// TwinCAT 3 PLC project PLC_MOTION
// Title: PLC_MOTION_LAYER
// Author: D. Hauer
// ProjectVersion: 01.00.34
// Description: MC-PtP, NCI, Camming cyclic execution layer for motion commands
// ProgramVersion: 3.1.4026.22
// libraries:
//   Tc2_EtherCAT, * (Beckhoff Automation GmbH)
//   Tc2_MC2, * (Beckhoff Automation GmbH)
//   Tc2_MC2_Camming, * (Beckhoff Automation GmbH)
//   Tc2_MC2_Drive, * (Beckhoff Automation GmbH)
//   Tc2_MC2_FlyingSaw, * (Beckhoff Automation GmbH)
//   Tc2_MC2_XFC, * (Beckhoff Automation GmbH)
//   Tc2_NCI, * (Beckhoff Automation GmbH)
//   Tc2_PlcInterpolation, * (Beckhoff Automation GmbH)
//   Tc2_Standard, * (Beckhoff Automation GmbH)
//   Tc2_System, * (Beckhoff Automation GmbH)
//   Tc2_Utilities, * (Beckhoff Automation GmbH)
//   Tc3_Module, * (Beckhoff Automation GmbH)
// project tree:
//   CAM/ CAM.TcPOU (not stored), GVL_CAM.TcGVL (not stored)
//   CAM/class/ FB_CamAxis.TcPOU (not stored), FB_CamCtrl.TcPOU, I_Cam_Ctrl.TcIO (not stored)
//   CAM/types/ ST_CAM_CTRL.TcDUT (not stored), ST_CAM_DATA.TcDUT (not stored), ST_CAM_INFO.TcDUT (not stored), ST_CAM_READ_VALUES_PARAMETER.TcDUT (not stored), ST_CAM_STATE.TcDUT (not stored), ST_CAM_OPTIONS.TcDUT (not stored), ST_CAM_SCALING_DATA.TcDUT (not stored), ST_MOTION_FUNCTION.TcDUT (not stored), ST_MOTION_FUNCTION_POINT.TcDUT
//   FLYING_SAW/class/ FB_FlyingBase.TcPOU (not stored), FB_FlyingCtrl.TcPOU (not stored), I_Fly_Ctrl.TcIO (not stored)
//   FLYING_SAW/ FLYING_SAW.TcPOU, GVL_FLYING_SAW.TcGVL
//   FLYING_SAW/types/ ST_FLY_CTRL.TcDUT (not stored), ST_FLY_DATA.TcDUT, ST_FLY_OPTIONS.TcDUT (not stored), ST_FLY_STATE.TcDUT (not stored), ST_FLY_SYNC_MODE.TcDUT (not stored)
//   FUNCTIONS/ FUNCTIONS.TcPOU (not stored), GVL_FUNCTIONS.TcGVL (not stored)
//   FUNCTIONS/TOUCH_PROBE/ FB_TouchProbe.TcPOU (not stored), I_TouchProbe.TcIO
//   FUNCTIONS/TOUCH_PROBE/types/ ST_2BIT.TcDUT (not stored), ST_CTRL_TOUCH_PROBE.TcDUT (not stored), ST_DC_Input.TcDUT (not stored), ST_MTI_INPUT.TcDUT (not stored), ST_MTI_STATUS.TcDUT (not stored), ST_STATE_TOUCH_PROBE.TcDUT (not stored)
//   FUNCTIONS/TRIGGER_BOX/ FB_TriggerBox.TcPOU (not stored), I_TriggerBox.TcIO (not stored)
//   FUNCTIONS/TRIGGER_BOX/types/ ST_CTRL_TRIGGER.TcDUT (not stored), ST_DC_Output.TcDUT (not stored), ST_DC_State.TcDUT (not stored), ST_STATE_TRIGGER.TcDUT (not stored), T_TriggerControlBits.TcDUT (not stored)
//   MAPPING/ MAPPING_AXIS_in.TcPOU (not stored), MAPPING_AXIS_out.TcPOU (not stored)
//   MAPPING/types/ U_AXIS_CTRL.TcDUT, U_AXIS_NC_PARAMETER_WRT.TcDUT (not stored), U_AXIS_HOMING.TcDUT (not stored), U_AXIS_MOTION_OPTIONS.TcDUT (not stored), U_AXIS_MOVE_DATA.TcDUT (not stored), U_AXIS_GEAR_IN.TcDUT (not stored), U_AXIS_NC_PARAMETER_RD.TcDUT (not stored), U_AXIS_STATE.TcDUT (not stored), U_AXIS_INFO.TcDUT (not stored), U_CAM_CTRL.TcDUT (not stored), U_CAM_DATA.TcDUT, U_CAM_INFO.TcDUT (not stored), U_CAM_STATE.TcDUT (not stored), U_FLY_CTRL.TcDUT (not stored), U_FLY_DATA.TcDUT (not stored), U_FLY_OPTIONS.TcDUT (not stored), U_FLY_STATE.TcDUT (not stored), U_NCI_AXIS_ID_GROUP.TcDUT (not stored), U_NCI_CTRL.TcDUT (not stored), U_NCI_INDEX_GROUP.TcDUT, U_NCI_R_PARAMETER_I.TcDUT (not stored), U_NCI_R_PARAMETER_Q.TcDUT (not stored), U_NCI_STATE.TcDUT, U_PARAMETER_SELECTOR_CTRL.TcDUT, U_PARAMETER_SELECTOR_STATE.TcDUT (not stored), U_TOUCH_PROBE_CTRL.TcDUT (not stored), U_TOUCH_PROBE_STATE.TcDUT (not stored), U_TRIGGER_CTRL.TcDUT (not stored), U_TRIGGER_STATE.TcDUT (not stored)
//   NCI/class/ FB_NciChannel.TcPOU (not stored), FB_NciChannelCtrl.TcPOU, I_NciChannel.TcIO (not stored), I_Nci_Ctrl.TcIO (not stored)
//   NCI/ GVL_NCI.TcGVL (not stored), NCI.TcPOU
//   NCI/types/ E_NCI_CTRL.TcDUT (not stored), E_NCI_CHANNEL_ERROR.TcDUT (not stored), E_NCI_STATE.TcDUT (not stored), E_NCI_INTERPRETER_STATE.TcDUT (not stored), ST_3D_Group.TcDUT (not stored), ST_NCI_CTRL.TcDUT (not stored), ST_NCI_M_FUNC.TcDUT (not stored), ST_Index_Group.TcDUT, ST_Interface_Group.TcDUT (not stored), ST_NciChannel_Ref.TcDUT (not stored), ST_NCI_STATE.TcDUT (not stored), ST_R_Parameter.TcDUT (not stored)
//   NC_PTP/class/ FB_McAxisBase.TcPOU, FB_McAxisCtrl.TcPOU, FB_ParameterSelector.TcPOU (not stored), I_McAxis.TcIO (not stored)
//   NC_PTP/ GVL_AXIS.TcGVL (not stored), MAIN_AXIS.TcPOU
//   NC_PTP/types/axis/ E_AxisEncoderType.TcDUT (not stored), ST_HomeParams.TcDUT (not stored)
//   NC_PTP/types/control/ E_AXIS_CTRL.TcDUT (not stored), E_AXIS_SELECTOR.TcDUT (not stored), E_AXIS_STATE.TcDUT, ST_AXIS_CTRL.TcDUT (not stored), ST_AXIS_INFO.TcDUT (not stored), ST_AXIS_LIMIT_SWITCHES.TcDUT (not stored), ST_AXIS_STATE.TcDUT (not stored), ST_GEAR_IN.TcDUT (not stored), ST_HOMING.TcDUT, ST_MOTION_OPTIONS.TcDUT (not stored), ST_MOVE_DATA.TcDUT (not stored), ST_NC_PARAMETER.TcDUT (not stored), ST_PARAMETER_SELECTOR_CTRL.TcDUT (not stored), ST_PARAMETER_SELECTOR_STATE.TcDUT (not stored)
//   XFC/ FB_Xfc.TcPOU
//   XFC/types/ E_XFC_CHECK.TcDUT (not stored)
//   XTS_TRANSPORT/MSG/ GVL_MSG.TcGVL (not stored)
//   _GVL/ GlobalTextList.TcGTLO (not stored), PLC_CONSTANT.TcGVL, PLC_VERSION.TcGVL
//   _MSG/ fb_LocalTime.TcPOU, fb_MessageData.TcPOU, fb_MessageDataCtrl.TcPOU, f_MessageSet.TcPOU (not stored), GVL_MSG_AXIS.TcGVL (not stored), I_MessageData.TcIO
//   _MSG/types/ e_Device.TcDUT, E_MessageType.TcDUT (not stored), E_MESSAGE_BATCH.TcDUT, E_MESSAGE_CHECK.TcDUT (not stored), E_MESSAGE_CTRL.TcDUT (not stored), E_MESSAGE_FLOW.TcDUT (not stored), E_MESSAGE_STATE.TcDUT, e_Subdevice.TcDUT, ST_Message.TcDUT (not stored), ST_MESSAGE_CTRL.TcDUT (not stored), ST_MESSAGE_STATE.TcDUT (not stored), TL_E_MESSAGETYPE.TcTLO (not stored)
//   / PlcTask.TcTTO, Visualization Manager.TcVMO (not stored)
//   _types/ E_CHECK_STATE.TcDUT (not stored), E_PROGRESS.TcDUT (not stored), f_GetProgress.TcPOU, f_GetState.TcPOU (not stored)
// real-time tasks:
//   TASK PlcTask: cycle T#1ms, priority 20, ADS port 350
//   TASK PlcTask1: cycle T#1ms, priority 1, ADS port 351
// motion (NC):
//   TASK NC-Task 1 SAF: cycle T#2ms, priority 4, ADS port 501
//   TASK NC-Task 1 SVB: cycle T#10ms, priority 8, ADS port 511
//   AXIS Axis 1 (id 1)
//     OtherSettings: AllowMotionCmdToSlave=true
//     encoder EncType=1
//     drive DrvType=5
//       Analog: TorqueSetpointScale=10, ScaleFactorActTorque=0.1
//       TimeComp: TaskDelayCycles=1
//     controller CtrType=1
//       CtrPara: PriorControlFactor=1
//         Observer: BandWidth=20
//   AXIS Axis 2 (id 2)
//     OtherSettings: AllowMotionCmdToSlave=true
//     encoder EncType=1
//     drive DrvType=5
//       Analog: TorqueSetpointScale=10, ScaleFactorActTorque=0.1
//       TimeComp: TaskDelayCycles=1
//     controller CtrType=1
//       CtrPara: PriorControlFactor=1
//         Observer: BandWidth=20
//   AXIS Axis 3 (id 3)
//     OtherSettings: AllowMotionCmdToSlave=true
//     encoder EncType=1
//     drive DrvType=5
//       Analog: TorqueSetpointScale=10, ScaleFactorActTorque=0.1
//       TimeComp: TaskDelayCycles=1
//     controller CtrType=1
//       CtrPara: PriorControlFactor=1
//         Observer: BandWidth=20
//   AXIS Axis 4 (id 4)
//     OtherSettings: AllowMotionCmdToSlave=true
//     encoder EncType=1
//     drive DrvType=5
//       Analog: TorqueSetpointScale=10, ScaleFactorActTorque=0.1
//       TimeComp: TaskDelayCycles=1
//     controller CtrType=1
//       CtrPara: PriorControlFactor=1
//         Observer: BandWidth=20
//   AXIS Axis 5 (id 5)
//     OtherSettings: AllowMotionCmdToSlave=true
//     encoder EncType=1
//     drive DrvType=5
//       Analog: TorqueSetpointScale=10, ScaleFactorActTorque=0.1
//       TimeComp: TaskDelayCycles=1
//     controller CtrType=1
//       CtrPara: PriorControlFactor=1
//         Observer: BandWidth=20
//   AXIS Axis 6 (id 6)
//     OtherSettings: AllowMotionCmdToSlave=true
//     encoder EncType=1
//     drive DrvType=5
//       Analog: TorqueSetpointScale=10, ScaleFactorActTorque=0.1
//       TimeComp: TaskDelayCycles=1
//     controller CtrType=1
//       CtrPara: PriorControlFactor=1
//         Observer: BandWidth=20
// variable links:
//   ExternControl/ExternControl Instance <-> PLC_MOTION/PLC_MOTION Instance
//     PlcTask Inputs/MAIN.eInitPlcMotion <-> PlcTask Outputs/MAIN_AXIS.eInit
//     PlcTask Inputs/MAPPING_in.AxisInfo.byState <-> PlcTask Outputs/MAPPING_AXIS_out.AxisInfo.byState
//     PlcTask Inputs/MAPPING_in.AxisParameterRd.byState <-> PlcTask Outputs/MAPPING_AXIS_out.AxisParameterOut.byState
//     PlcTask Inputs/MAPPING_in.AxisState.byState <-> PlcTask Outputs/MAPPING_AXIS_out.AxisState.byState
//     PlcTask Outputs/MAPPING_out.AxisCtrl.byCtrl <-> PlcTask Inputs/MAPPING_AXIS_in.AxisCtrl.byCtrl
//     PlcTask Outputs/MAPPING_out.AxisGearInData.byCtrl <-> PlcTask Inputs/MAPPING_AXIS_in.AxisGearInData.byCtrl
//     PlcTask Outputs/MAPPING_out.AxisHoming.byCtrl <-> PlcTask Inputs/MAPPING_AXIS_in.AxisHoming.byCtrl
//     PlcTask Outputs/MAPPING_out.AxisMotionOptions.byCtrl <-> PlcTask Inputs/MAPPING_AXIS_in.AxisMotionOptions.byCtrl
//     PlcTask Outputs/MAPPING_out.AxisMoveData.byCtrl <-> PlcTask Inputs/MAPPING_AXIS_in.AxisMoveData.byCtrl
//     PlcTask Outputs/MAPPING_out.AxisParameterWrt.byCtrl <-> PlcTask Inputs/MAPPING_AXIS_in.AxisParameterIn.byCtrl
//   PLC_MOTION/PLC_MOTION Instance <-> NC-Task 1 SAF/Axes/Axis 1
//     PlcTask Inputs/GVL_AXIS.AxisRef[1].NcToPlc <-> Outputs/ToPlc
//     PlcTask Outputs/GVL_AXIS.AxisRef[1].PlcToNc <-> Inputs/FromPlc
//   PLC_MOTION/PLC_MOTION Instance <-> NC-Task 1 SAF/Axes/Axis 2
//     PlcTask Inputs/GVL_AXIS.AxisRef[2].NcToPlc <-> Outputs/ToPlc
//     PlcTask Outputs/GVL_AXIS.AxisRef[2].PlcToNc <-> Inputs/FromPlc
//   PLC_MOTION/PLC_MOTION Instance <-> NC-Task 1 SAF/Axes/Axis 3
//     PlcTask Inputs/GVL_AXIS.AxisRef[3].NcToPlc <-> Outputs/ToPlc
//     PlcTask Outputs/GVL_AXIS.AxisRef[3].PlcToNc <-> Inputs/FromPlc
//   PLC_MOTION/PLC_MOTION Instance <-> NC-Task 1 SAF/Axes/Axis 4
//     PlcTask Inputs/GVL_AXIS.AxisRef[4].NcToPlc <-> Outputs/ToPlc
//     PlcTask Outputs/GVL_AXIS.AxisRef[4].PlcToNc <-> Inputs/FromPlc
//   PLC_MOTION/PLC_MOTION Instance <-> NC-Task 1 SAF/Axes/Axis 5
//     PlcTask Inputs/GVL_AXIS.AxisRef[5].NcToPlc <-> Outputs/ToPlc
//     PlcTask Outputs/GVL_AXIS.AxisRef[5].PlcToNc <-> Inputs/FromPlc
//   PLC_MOTION/PLC_MOTION Instance <-> NC-Task 1 SAF/Axes/Axis 6
//     PlcTask Inputs/GVL_AXIS.AxisRef[6].NcToPlc <-> Outputs/ToPlc
//     PlcTask Outputs/GVL_AXIS.AxisRef[6].PlcToNc <-> Inputs/FromPlc

CONFIGURATION PLC_MOTION
    RESOURCE PLC ON TwinCAT3
        TASK PlcTask(INTERVAL := T#1ms, PRIORITY := 1);
        PROGRAM MAPPING_AXIS_in WITH PlcTask : MAPPING_AXIS_in;
        PROGRAM MAIN_AXIS WITH PlcTask : MAIN_AXIS;
        PROGRAM FUNCTIONS WITH PlcTask : FUNCTIONS;
        PROGRAM NCI WITH PlcTask : NCI;
        PROGRAM CAM WITH PlcTask : CAM;
        PROGRAM FLYING_SAW WITH PlcTask : FLYING_SAW;
        PROGRAM MAPPING_AXIS_out WITH PlcTask : MAPPING_AXIS_out;
    END_RESOURCE
END_CONFIGURATION

// ---- CAM/types/ST_MOTION_FUNCTION_POINT.TcDUT
{attribute 'pack_mode' := '2'}
TYPE ST_MOTION_FUNCTION_POINT :
STRUCT
   nPointIndex            : UINT;
   nFunctionType          : UINT;
   wPointType             : WORD;
   nRelIndexNextPoint     : UINT;
   rMasterPos             : LREAL; (* X *)
   rSlavePos              : LREAL; (* Y *)
   rSlaveVelo             : LREAL; (* Y' *)
   rSlaveAcc              : LREAL; (* Y'' *)
   rSlaveJerk             : LREAL; (* Y''' *)
END_STRUCT
END_TYPE

// ---- FLYING_SAW/types/ST_FLY_DATA.TcDUT
{attribute 'pack_mode' := '2'}
TYPE ST_FLY_DATA :
STRUCT
  rDeltaToMasterPos       : LREAL;
  rModuloSyncPosSlave     : LREAL;
  rMasterStartDistance    : LREAL;
  rDelta                  : LREAL  := 0.1;
  rGearNumerator          : LREAL;
  iGearDenumerator        : USINT  := 1;
  nMasterAxisId           : UDINT; // NC axis ID, index is looked up by Cmd
  rModulo                 : lreal; // float for modulo calculation, this is independent of the NC on purpose, you may connect the modulo divisor from the NC on the outside of the FlyingSaw class
END_STRUCT
END_TYPE

// ---- MAPPING/types/U_AXIS_CTRL.TcDUT
TYPE U_AXIS_CTRL :
UNION

  stCtrl              : ARRAY[1..MAX_AXIS] OF ST_AXIS_CTRL;

  byCtrl    AT %I*    : ARRAY[1..MAX_AXIS] OF
                        ARRAY[1..SIZEOF(ST_AXIS_CTRL)] OF BYTE;
END_UNION
END_TYPE

// ---- MAPPING/types/U_CAM_DATA.TcDUT
TYPE U_CAM_DATA :
UNION
  stCtrl              : ARRAY[1..MAX_AXIS] OF ST_CAM_DATA;

  byCtrl    AT %I*    : ARRAY[1..MAX_AXIS] OF
                        ARRAY[1..SIZEOF(ST_CAM_DATA)] OF BYTE;
END_UNION
END_TYPE

// ---- MAPPING/types/U_NCI_INDEX_GROUP.TcDUT
TYPE U_NCI_INDEX_GROUP :
UNION

  stCtrl              : ARRAY[1..MAX_NCI_CH] OF ST_Index_Group;

  byCtrl    AT %I*    : ARRAY[1..MAX_NCI_CH] OF
                        ARRAY[1..SIZEOF(ST_Index_Group)] OF BYTE;
END_UNION
END_TYPE

// ---- MAPPING/types/U_NCI_STATE.TcDUT
TYPE U_NCI_STATE :
UNION

  stState             : ARRAY[1..MAX_NCI_CH] OF ST_NCI_STATE;

  byState   AT %Q*    : ARRAY[1..MAX_NCI_CH] OF
                        ARRAY[1..SIZEOF(ST_NCI_STATE)] OF BYTE;
END_UNION
END_TYPE

// ---- MAPPING/types/U_PARAMETER_SELECTOR_CTRL.TcDUT
TYPE U_PARAMETER_SELECTOR_CTRL :
UNION
  stCtrl              : ST_PARAMETER_SELECTOR_CTRL;

  byCtrl    AT %I*    : ARRAY[1..SIZEOF(ST_PARAMETER_SELECTOR_CTRL)] OF BYTE;

END_UNION
END_TYPE

// ---- NCI/types/ST_Index_Group.TcDUT
{attribute 'pack_mode' := '2'}
TYPE ST_Index_Group :
STRUCT
  nXAxisIdx     : UDINT := 1;
  nYAxisIdx     : UDINT := 2;
  nZAxisIdx     : UDINT := 3;

  nQ1AxisIdx    : UDINT;
  nQ2AxisIdx    : UDINT;
  nQ3AxisIdx    : UDINT;
  nQ4AxisIdx    : UDINT;
  nQ5AxisIdx    : UDINT;
END_STRUCT
END_TYPE

// ---- NC_PTP/types/control/E_AXIS_STATE.TcDUT
{attribute 'qualified_only'}
{attribute 'to_string'}
TYPE E_AXIS_STATE :
(
  AXIS_NULL,   // null reaction to command
  AXIS_INIT,
  AXIS_DISABLE,
  AXIS_ENABLE,

  AXIS_NO_INIT  := 9,
  
  AXIS_IDLE     := 10, // clear axis and enable
  AXIS_HOME,
  AXIS_MOVE_POS,
  AXIS_MOVE_VELO,
  AXIS_HALT,
  AXIS_STOP,
  AXIS_SEND_TO_POS,

  AXIS_RESET              := 19,
  AXIS_STARTUP            := 20,

  AXIS_MOVE_BUFFER        := 30,
  AXIS_MOVE_BUFFER_VELO,

  AXIS_PARAMETER_READ     := 40, // command for reading and writing parameter
  AXIS_PARAMETER_WRITE,
  AXIS_PARAMETER_WRITE_PERSISTENT,


  AXIS_GEAR_IN            := 50,
  AXIS_GEAR_OUT,
  AXIS_GEAR_IN_MULTIMASTER,

  CAM_INIT                := 60,
  CAM_IN,
  CAM_OUT,
  CAM_SCALING,
  CAM_INFO,
  CAM_RD_MOTION_FUNCTION,
  CAM_RD_MOTION_FUNCTION_POINT,
  CAM_RD_MOTION_FUNCTIONS_VALUES,
  CAM_WRT_MOTION_FUNCTION,
  CAM_WRT_MOTION_FUNCTION_POINT

)UINT;
END_TYPE

// ---- NC_PTP/types/control/ST_HOMING.TcDUT
{attribute 'pack_mode' := '2'}
TYPE ST_HOMING :
STRUCT
  bExecute      : BIT;

  stHomingParam : ST_HomeParams;
END_STRUCT
END_TYPE

// ---- _MSG/types/e_Device.TcDUT
{attribute 'to_string'}
TYPE e_Device :
(
  // txt file logging LOG_FILE
  Device_Null,                  // NULL               - not to be used
  Device_Main,                  // MAIN(PRG)          - reserved for MAIN(PRG)
  Device_Nci,                   // NCI(PRG)           - reserved for NCI(PRG)
  Device_Cam,                   // CAM(PRG            - reserved for CAM(PRG)
  Device_Functions,             // FUNCTIONS(PRG)     - reserved for FUNCTIONS(PRG)
  Device_FlyingSaw,             // FLYING_SAW(PRG)    - reserved for FLYING_SAW(PRG)
  Device_MainApplication,       // MAIN_APP(PRG)

  Device_ParameterSelector,     // fb_ParameterSelector can only exist once in a project.
  Device_Configuration,         // fb_Configuration can handle multiple files therefore only one instance is required
  Device_XmlData,               // generic XML Data (e.g. persistent data)
  Device_Utilities,             // service calls to anyone you may want to talk to, the main intent is to get XPU and TcXtsIo data to the application side


  General           :=  1000,
  CaGroup           :=  2000,
  Xpu               :=  3000,
  XpuCtrl           :=  4000,
  Mover             :=  5000,
  MoverCtrl         :=  6000,
  XtsTransportUnit  :=  7000,
  XfcTriggerBox     :=  8000,
  XfcTouchProbe     :=  9000,
  XtsStation        := 10000,

  Camming           := 11000,
  NciChannel        := 12000,
  NciChannelCtrl    := 13000,
  Axis              := 14000,
  XfcAxis           := 15000,

  // txt file logging LOG_FILE_METRICS
  Metrics           := 16000,

  FlyingSaw         := 17000,


  // txt file logging LOG_FILE_APP
  Process           := 20000,
  ProcessListCtrl   := 21000,
  TicketListCtrl    := 22000,

  Application       := 30000,

  // txt file logging LOG_FILE_PRODUCT - this is for you to use
  DataProduct       := 40000
)UDINT;
END_TYPE

// ---- _MSG/types/E_MESSAGE_BATCH.TcDUT
{attribute 'qualified_only'}
{attribute 'strict'}
{attribute 'to_string'}
TYPE E_MESSAGE_BATCH :
(
	MSG_BATCH_NULL,
  MSG_BATCH_JOB_STARTED,
  MSG_BATCH_NEXT_IN_JOB,
  MSG_BATCH_JOB_DONE
)UINT;
END_TYPE

// ---- _MSG/types/E_MESSAGE_STATE.TcDUT
{attribute 'qualified_only'}
//{attribute 'strict'}
{attribute 'to_string'}
TYPE E_MESSAGE_STATE :
(
	MSG_STATE_NULL,
  MSG_STATE_INIT    := 10,
  MSG_STATE_IDLE    := 30,
  MSG_STATE_WRITE   := 50
)UINT;
END_TYPE

// ---- _MSG/types/e_Subdevice.TcDUT
{attribute 'strict'}
{attribute 'to_string'}
TYPE e_Subdevice :
(
  // sub device for message system
  General                 :=  0,
  MainInit,
  // Motion Control FB Instances
  fbPower,
  fbReset,
  fbResetSercos,
  fbHalt,
  fbStop,                 // 5
  fbHome,
  fbJog,
  fbMoveVelocity1,
  fbMoveVelocity2,
  fbMoveAbsolute1,        // 10
  fbMoveAbsolute2,
  fbMoveEndless,
  fbMovePtP,
  fbMoveVelo,

  // CA CollisionAvoidance FB instances
  // CA group fb instances
  fbCaGroup             := 30,
  fbMoveToPosCa,
  fbSendToAbsPosCa,
  fbSendToModuloPosCa,
  fbGearInPosCa,
  fbGroupAddAxis,
  fbGroupRemoveAxis,
  fbGroupDisable,
  fbGroupEnable,
  fbGroupErrorRead,
  fbGroupStatusRead,
  fbGroupReset,
  fbGroupStop,
  fbHaltCa,
  fbSendToPos,

  fbGearIn                := 50,
  fbGearOut,
  fbGearInMultiMaster,

  fbGearInPos,
  fbGearInVelo,


  fbCamOut                := 80,
  fbCamInV2,
  fbCamScalingV2,
  fbCamInfoV2,
  fbReadMotionFunction,
  fbReadMotionFunctionPoint,
  fbReadMotionFunctionValues,
  fbWriteMotionFunction,
  fbWriteMotionFunctionPoint,
  fbSetOnlineChangeMode,

  fbReadParameter         := 100,
  fbReadBoolParameter,
  fbWriteParameter,
  fbWriteBoolParameter,
  fbWriteParameterPersistent,

  fbBuildGroup            := 200,
  fbClearGroup,
  fbLoadProg,
  fbResetItp,
  fbStartStopItp,
  fbEStopItp,             // 205
  fbStepOnAfterEStopItp,
  fbConfirmHskItp,
  fbDelDtgItp,
  fbNciFeedTablePreparation,
  fbNciFeedTable,         // 210
  fbReadLine,
  fbItpReadRParams,
  fbItpWriteRParams,
  Get_ItpState,
  Get_Error,              // 215


  XfcPositionAtTime       := 300,
  XfcTimeOfPosition,
  XfcTimeToPosition,
  XfcTimeToModuloPosition,
  XfcRecordedPosition,
  XfcTouchProbe,          // 305
  XfcTouchProbeEL1258,
  XfcTouchProbeOptions,
  XfcTriggerRef,
  XfcTriggerRef_MT,
  XfcEl1258Interface_MT,  // 310
  XfcRecordedPosition_MT,
  XfcTriggerOut,
  XfcTriggerStart,
  XfcSwitchOn_2252,
  XfcSwitchOff_2252,      // 315
  XfcInit,
  XfcLatchPosition,
  XfcWaitForPosition,

  AxisMode              := 1000,
  AxisControl,
  AxisStartUp,
  AxisCycle,
  AxisIdle,

  NciControl            := 2000,
  NciStartUp,
  NciCycle,
  NciIdle,

  FlyingSawControl      := 2100,
  FlyingSawStartUp,


  StationLinkedList     := 3000,
  StationInitList,
  StationAddHead,
  StationAddTail,
  StationGetHead,
  StationRemoveHeadValue,
  StationGearInDistanceToSync,
  StationGearInSyncStart,
  StationGearInSyncMove,
  StationGearInSyncEnd,
  StationCalcInfeedPosition,

  StationControl        := 4000,
  StationState, 

  Xpu_fbEnvironment     := 5000,
  Xpu_fbProcessingUnit,
  Xpu_fbXpuPart,
  Xpu_fbXpuTrack,
  Xpu_fbMc2CaGroup,
  Xpu_fbParameterSet,
  Xpu_fbNctController,

  Xpu_fbPartModules     := 5500,

  Xpu_fbMoverXpu        := 6000,

  Xpu_fbNctBaseUnit     := 6500,

  TransportUnit_General := 7000,
  TransportUnit_Restart := 7010,
  TransportUnit_Start,
  TransportUnit_XpuInit,
  TransportUnit_StationClearOutfeed,

  CamControl            := 8000,
  CamStartUp,
  CamCycle,

  Process_StationCollector    := 11000,
  Process_ProcessCollector    := 11100,
  Process_ProcessCollector_Init,
  Process_ProcessCollector_Cycle,
  Process_ProcessCollector_Control,

  Process_LinkedList_GetHead,
  Process_LinkedList_RemoveHead,
  Process_LinkedList_AddTail,
  Process_LinkedList_CheckData,
  Process_StationQueue_Check,

  Process_LinkedList_Com              := 11200,
  Process_LinkedList_Com_Init,
  Process_LinkedList_Com_Cmd,
  Process_LinkedList_Com_AddHead,
  Process_LinkedList_Com_AddTail,
  Process_LinkedList_Com_DelHead,
  Process_LinkedList_Com_DelTail,
  Process_LinkedList_Com_GetHead,
  Process_LinkedList_Com_GetTail,


  Instance_Command              := 12000,
  Instance_ProcessConductor,
  Instance_BufferInfeed,
  Instance_Infeed,
  Instance_BufferOutfeed,
  Instance_Outfeed,
  Instance_Sender_Buffer,

  Ticket_LinkedList_Ctrl        := 12100,
  Ticket_LinkedList_Com_Init,
  Ticket_LinkedList_Com_Cmd,
  Ticket_LinkedList_Com_AddHead,
  Ticket_LinkedList_Com_AddTail,
  Ticket_LinkedList_Com_DelHead,
  Ticket_LinkedList_Com_DelTail,
  Ticket_LinkedList_Com_GetHead,
  Ticket_LinkedList_Com_GetTail,
  

  Application                 := 13000,
  Application_Check,
  Application_Clear,
  Application_Cmd,
  Application_Disable,
  Application_Enable,
  Application_Finish,
  Application_Init,
  Application_Proceed,
  Application_Work


)DINT;
END_TYPE

// ---- FLYING_SAW/GVL_FLYING_SAW.TcGVL
{attribute 'qualified_only'}
VAR_GLOBAL
  //-----------------------------------------------------------------------------
  // command and state structure
  //  - datafields for anyone to access
  //    - ADS via symbol
  //    - cyclic mapping to any other cyclic network/runtime
  //-----------------------------------------------------------------------------
  Ctrl                        : ARRAY[1..PLC_CONSTANT.MAX_AXIS] OF ST_FLY_CTRL;      // command structure to write into
  State                       : ARRAY[1..PLC_CONSTANT.MAX_AXIS] OF ST_FLY_STATE;     // state structure to read from


  //-----------------------------------------------------------------------------
  // data and info structure
  //  - parameter data fields for
  //    - Ctrl  --> Data
  //    - State --> Info
  //-----------------------------------------------------------------------------
//  Info                        : ARRAY[1..PLC_CONSTANT.MAX_AXIS] OF ST_FLY_INFO;
  Data                        : ARRAY[1..PLC_CONSTANT.MAX_AXIS] OF ST_FLY_DATA;


  //-----------------------------------------------------------------------------
  // R/W datafields
  // - optional data for CheckMask
  // - The Options contains two position values as limits. 
  //   The check for these position limits can be activated. 
  //   To do this, two flags 
  //   (GearInSync_CheckMask_OptionalMinPos, 
  //    GearInSync_CheckMask_OptionalMaxPos) 
  //   have to be set in the SyncMode structure.
  //
  //-----------------------------------------------------------------------------
  Options                     : ARRAY[1..PLC_CONSTANT.MAX_AXIS] OF ST_FLY_OPTIONS;


  //-----------------------------------------------------------------------------
  // cyclic interface function block: FB_FlyingCtrl
  //  - Tc2_MC2_FlyingSaw functions are here 
  //-----------------------------------------------------------------------------
{IF defined (SAW)}
  {info 'PLC_MOTION_LAYER: FLYING_SAW'}
  Control                     : ARRAY[1..PLC_CONSTANT.MAX_AXIS] OF FB_FlyingCtrl;
{ELSE}
  Control                     : ARRAY[1..PLC_CONSTANT.MAX_AXIS] OF I_Fly_Ctrl;
{END_IF}

END_VAR

// ---- _GVL/PLC_CONSTANT.TcGVL
//{attribute 'qualified_only'}
VAR_GLOBAL CONSTANT


  //-----------------------------------------------------------------------------
  // AXIS related limits
  //-----------------------------------------------------------------------------
  MAX_AXIS              : UINT    := 6;
  MAX_RETRY             : UINT    := 5;


  //-----------------------------------------------------------------------------
  // NCI related limits and *.nc standard folder
  //-----------------------------------------------------------------------------
{IF NOT defined (BSD)}
  NCI_DIR               : STRING  := 'C:\TwinCAT\Mc\Nci\';
{ELSE}
  NCI_DIR               : STRING  := '/usr/local/etc/TwinCAT/Mc/Nci/';
{END_IF}

{IF defined (NCI)}
  {info 'PLC_MOTION_LAYER: NCI'}
  NCI_ACTIVE            : BOOL    := TRUE;
  CONFIG_NAME           : STRING  := 'NCI_Spec_Ch_';
{ELSE}
  NCI_ACTIVE            : BOOL    := FALSE;
  CONFIG_NAME           : STRING  := 'NCI_NOT_ACTIVE';
{END_IF}

  MAX_NCI_CH            : UINT    := 1;

  MAX_PATH_STEPS        : UINT    := 5;
  MAX_MC_AXIS           : UINT    := 3;
  MAX_AUX_AXIS          : UINT    := 2;
  MAX_R_PARA            : UINT    := 10;


  //-----------------------------------------------------------------------------
  // CAMMING related limits
  //-----------------------------------------------------------------------------
{IF defined (CAM)}
  {info 'PLC_MOTION_LAYER: CAM'}
  CAM_ACTIVE                  : BOOL    := TRUE;
{ELSE}
  CAM_ACTIVE                  : BOOL    := FALSE;
{END_IF}

  MAX_CAM_CH                  : UINT    := 1;

  MAX_MOTION_FUNCTION_POINTS  : UINT    := 10;

  // HAUD
  // 17.07.2024
  // Start Implementation of Position Trigger function
  //  - Timestamp/position output
  //  - Latch DC time from input
  
  MAX_TRIGGER_BOX             : UINT := 12;
  MAX_TOUCH_PROBE             : UINT := 12;
  MAX_TRIGGER_COUNT           : UINT :=  4;
  MAX_MTI_CH                  : UINT :=  1; // MAX mti channel per EL terminal

{IF defined (XFC)}
  {info 'PLC_MOTION_LAYER: XFC'}
  XFC_ACTIVE                  : BOOL := TRUE;
{ELSE}
  XFC_ACTIVE                  : BOOL := FALSE;
{END_IF}

  // HAUD
  // 2026 05 28
  // Gear In Pos implementation for flying saw application 

{IF defined (SAW)}
  {info 'PLC_MOTION_LAYER: FLYING_SAW'}
  FLY_SAW_ACTIVE              : BOOL  := TRUE;
{ELSE}
  FLY_SAW_ACTIVE              : BOOL  := FALSE;
{END_IF}
END_VAR

// ---- _GVL/PLC_VERSION.TcGVL
{attribute 'qualified_only'}
VAR_GLOBAL CONSTANT
  VERSION               : STRING := 'V 01.00.38';

  // 2025 05 28 HAUD
  // Flying Saw wrapper

  // 2025 05 13 HAUD
  //
  // FB_McAxisBase.MoveVeloBuffer Test, changes for setpoint change detection

  // 2025 10 24 HAUD
  //
  // documentation added, 
  // project dev changed to 4026.19
  // Ambiguities resoved

  // 2025 08 21 HAUD
  //
  // e_Device: Application added
  // e_Subdevices: merge with XTS_TRANSPORT_LAYER
  // FB_McAxis: testing SendToPos, distance added to method interface

  // 2025 02 17 HAUD
  //
  // code review
  // Message Levels are set during initialization
  // sizeof mapping data is fetched at startup only

  // 2025 01 09 HAUD
  //
  // - FUNCTIONS
  //    - code review
  //    - ctrl/state mechanic harmonized
  // - MAPPING
  //    - UNIONS added

  // 2024 08 08 HAUD
  //
  // - TC_PLC_MOTION_LAYER: 
  //    - XFC base class added
  //    - TriggerBox (DC output set, DC Input latch)
  //    - TouchProbe (DC Input latch: positive, negative)

  // 2024 06 21 HAUD
  //
  // - TC_PLC_MOTION_LAYER: 
  //    - E_PROGRESS refactoring to match TC_XTS_TRANSPORT_LAYER
  

  // 2024 06 10 HAUD
  //
  // - TC_PLC_MOTION_LAYER: 
  //    - rename repository
  //    - remove LEGACY compatibility
  //
  // - PLC_OPEN_DRIVE:
  //    - deprecated


  // 2024 05 31 HAUD
  // 
  // V 01.00.02
  // precompiler defines: 
  //  - BSD: 
  //    - Tc-BSD file system is used else Windows file system is used
  //
  //  - TEST:
  //    - GVL_MSG.MessageLevel
  // Axis, Cam, Nci have individual message levels now

  // 2024 03 09 HAUD
  // 
  // V 01.00.01
  // MC PtP - execution layer with optional mapping
  // NCI    - execution layer with optional mapping
  // CAM    . execution layer with optional mapping
  // precompiler defines: 
  //  - WIN: windows file system is used else Tc-BSD file system is used
  //  - NCI: NCI libraries are linked in project
  //  - CAM: Camming libraries are linked in project
  //  - AXIS_MAP: mapping is used


  // 2024 02 15 HAUD
  // 
  // V 00.50.04
  //
  // Buffered moves test
  // CamIn Test --> TODO MultiCam
  // Message system, cyclic check for write
  

  // 2024 01 12 HAUD
  //
  // V 00.50.03
  //
  // Building is done
  // start of UnitTesting

  // 2024 01 17 HAUD
  //
  // V 00.50.02
  // 
  // start camming implementation (MC_CamIn_V2)
  // legacy namespace available for downward compatibility of ADS Symbol names

  // 2023 12 23 HAUD
  // NC_PTP
  // - redesign for PLC_OPEN_DRIVE started 
  //    --> E_PROGRESS for state feedback
  // - FB_AxisControl inherits FB_McAxis


  //  2023 10 19
  //  HAUD
  // first draft 
  // TODO: everything

END_VAR

// ---- FUNCTIONS/TOUCH_PROBE/I_TouchProbe.TcIO
INTERFACE I_TouchProbe

PROPERTY Ctrl : REFERENCE TO ARRAY [1..MAX_TOUCH_PROBE] OF ST_CTRL_TOUCH_PROBE
SET
END_SET
END_PROPERTY

METHOD Cycle : BOOL
VAR_INPUT
END_VAR
END_METHOD

PROPERTY Index : udint
GET
END_GET
SET
END_SET
END_PROPERTY

PROPERTY Input : pointer TO ARRAY [1..MAX_TOUCH_PROBE] OF ST_MTI_Input
SET
END_SET
END_PROPERTY

PROPERTY InputState : pointer TO ARRAY [1..MAX_TOUCH_PROBE] OF ST_MTI_STATUS
SET
END_SET
END_PROPERTY

PROPERTY ItfAxis : ARRAY[1..MAX_AXIS]       OF I_McAxis
SET
END_SET
END_PROPERTY

PROPERTY MessageLevel : e_messagetype
GET
END_GET
SET
END_SET
END_PROPERTY

PROPERTY State :  REFERENCE TO ARRAY[1..MAX_TOUCH_PROBE] OF ST_STATE_TOUCH_PROBE;
SET
END_SET
END_PROPERTY

END_INTERFACE

// ---- _MSG/I_MessageData.TcIO
INTERFACE I_MessageData

PROPERTY DirRoot : POINTER to string(255)
SET
END_SET
END_PROPERTY

PROPERTY ErrorIndex : reference to uint
SET
END_SET
END_PROPERTY

PROPERTY FileRoot : pointer to string(255)
SET
END_SET
END_PROPERTY

PROPERTY LocalTime : pointer to DT
SET
END_SET
END_PROPERTY

PROPERTY MessageIndex : reference to uint
SET
END_SET
END_PROPERTY

PROPERTY MsgList : pointer to ARRAY[1..GVL_MSG.MAX_MESSAGE] OF st_message
SET
END_SET
END_PROPERTY

END_INTERFACE

// ---- NC_PTP/MAIN_AXIS.TcPOU
PROGRAM MAIN_AXIS
VAR
  eInit         AT %Q*      : E_PROGRESS;   // shall be checked by controlling entity, before using Ctrl/State structs

  nAxis,
  nAxisInit                 : UINT;

  stMsg                   : ST_Message;
  eMsgState               : e_message_state;
  eMsgProgress            : E_PROGRESS;
  eMtrState               : e_message_state;
  eMtrProgress            : E_PROGRESS;

  tIdleWriteMotion        : TIME := T#5S;
  tIdleWriteMetric        : TIME := T#5S;
  tonIdleWriteMotion      : Tc2_Standard.TON;
  tonIdleWriteMetric      : Tc2_Standard.TON;
END_VAR

//-----------------------------------------------------------------------------------------------------------------
// Local time; used for timestamps
//-----------------------------------------------------------------------------------------------------------------
GVL_MSG_AXIS.fbLocalTime();
GVL_MSG.sLocalTime                            :=
GVL_MSG_AXIS.sLocalTime                       := GVL_MSG_AXIS.fbLocalTime.LocalTimeString;
GVL_MSG.dtLocalTime                           :=
GVL_MSG_AXIS.dtLocalTime                      := GVL_MSG_AXIS.fbLocalTime.LocalTime;
//-----------------------------------------------------------------------------------------------------------------
// /assign dataflow
//-----------------------------------------------------------------------------------------------------------------
FOR nAxis := 1 TO PLC_CONSTANT.MAX_AXIS
DO
  GVL_AXIS.Control[nAxis].AxisIndex           := nAxis;
  GVL_AXIS.Control[nAxis].MessageLevel        := GVL_MSG_AXIS.MessageLevelAxisPtp[nAxis];

  GVL_AXIS.Control[nAxis].AxisCtrl            := ADR(GVL_AXIS.Ctrl);          // command
  GVL_AXIS.Control[nAxis].AxisState           := ADR(GVL_AXIS.State);         // state + result of command

  GVL_AXIS.Control[nAxis].Axes                REF=   GVL_AXIS.AxisRef;        // All for one; coupling requires access across all axes

  GVL_AXIS.Control[nAxis].AxisInfo            := ADR(GVL_AXIS.Info);          // axis information: act/set values and bits from axis
  GVL_AXIS.Control[nAxis].AxisData            := ADR(GVL_AXIS.Data);          // position and dynamic constraints for movement
  GVL_AXIS.Control[nAxis].AxisGearInParameter := ADR(GVL_AXIS.GearInParameter);

  GVL_AXIS.Control[nAxis].NcParameterOut      := ADR(GVL_AXIS.NcParameterOut);
  GVL_AXIS.Control[nAxis].NcParameterIn       := ADR(GVL_AXIS.NcParameterIn);

  GVL_AXIS.Control[nAxis].HomingParameter     := ADR(GVL_AXIS.HomeParameter);
  GVL_AXIS.Control[nAxis].MotionOptions       := ADR(GVL_AXIS.MotionOptions);
  GVL_AXIS.Control[nAxis].LimitSwitches       := ADR(GVL_AXIS.LimitSwitches);

  GVL_AXIS.ItfMcAxis[nAxis]                   := GVL_AXIS.Control[nAxis]; 
END_FOR

GVL_AXIS.ParameterSelector.MessageLevel       :=   GVL_MSG.MessageLevel;
GVL_AXIS.ParameterSelector.Ctrl               REF= GVL_AXIS.SelectorCtrl;
GVL_AXIS.ParameterSelector.State              REF= GVL_AXIS.SelectorState;
GVL_AXIS.ParameterSelector.ItfAxis            REF= GVL_AXIS.ItfMcAxis;
//-----------------------------------------------------------------------------------------------------------------
// assign dataflow/
//-----------------------------------------------------------------------------------------------------------------
//-----------------------------------------------------------------------------------------------------------------
//-----------------------------------------------------------------------------------------------------------------
// /INIT
// - successful init is required for other optional members to start
//-----------------------------------------------------------------------------------------------------------------
CASE eInit
OF
  E_PROGRESS.PROGRESS_INVALID:
    GVL_MSG_AXIS.MotionMessageCtrl.Cmd        := E_MESSAGE_CTRL.MSG_CTRL_NULL;
    GVL_MSG_AXIS.MetricMessageCtrl.Cmd        := E_MESSAGE_CTRL.MSG_CTRL_NULL;

    FOR nAxis := 1 TO PLC_CONSTANT.MAX_AXIS
    DO
      GVL_MSG_AXIS.MessageLevelAxisPtp[nAxis] := E_MessageType.eMessageVerbose; //GVL_MSG.MessageLevel;
    END_FOR
    nAxisInit                                 := 1;
    eInit                                     := E_PROGRESS.PROGRESS_INIT;
  //-----------------------------------------------------------------------------
  //-----------------------------------------------------------------------------
  E_PROGRESS.PROGRESS_INIT:
    stMsg.eType                               := E_MessageType.eMessageInfo;
    stMsg.eDevice                             := e_Device.Device_MainAxis;
    stMsg.eSubdevice                          := e_SubDevice.MainInit;
    stMsg.iErrorNumber                        := MAX_AXIS;
    stMsg.sText                               := concat('MAIN_AXIS.eInit: ', TO_STRING(eInit));
    f_MessageSet(stMsg);

    GVL_MSG_AXIS.MotionMessageCtrl.Cmd        := E_MESSAGE_CTRL.MSG_CTRL_INIT;
    GVL_MSG_AXIS.MetricMessageCtrl.Cmd        := E_MESSAGE_CTRL.MSG_CTRL_INIT;
    eInit                                     := E_PROGRESS.PROGRESS_BUSY;
  //-----------------------------------------------------------------------------
  //-----------------------------------------------------------------------------
  E_PROGRESS.PROGRESS_BUSY:
    eInit                                     := E_PROGRESS.PROGRESS_PREPARE;
  //-----------------------------------------------------------------------------
  //-----------------------------------------------------------------------------
  E_PROGRESS.PROGRESS_PREPARE:
    stMsg.eType                               := E_MessageType.eMessageVerbose;
    stMsg.eDevice                             := e_Device.Device_MainAxis;
    stMsg.eSubdevice                          := e_SubDevice.MainInit;
    stMsg.iErrorNumber                        := nAxisInit;
    stMsg.sText                               := concat('AxisInit Index: ', TO_STRING(nAxisInit));

    IF (GVL_MSG_AXIS.MessageLevelAxisPtp[nAxisInit] = E_MessageType.eMessageVerbose)
    THEN
      f_MessageSet(stMsg);
    END_IF

    GVL_AXIS.Ctrl[nAxisInit].eCmd             := E_AXIS_CTRL.AXIS_NULL;
    eInit                                     := E_PROGRESS.PROGRESS_STARTUP;
  //-----------------------------------------------------------------------------
  //-----------------------------------------------------------------------------
  E_PROGRESS.PROGRESS_STARTUP:
    GVL_AXIS.Ctrl[nAxisInit].eCmd             := E_AXIS_CTRL.AXIS_INIT;

    IF    (GVL_AXIS.State[nAxisInit].eState = E_AXIS_STATE.AXIS_INIT + E_PROGRESS.PROGRESS_ERROR)
    THEN
      eInit                                   := E_PROGRESS.PROGRESS_ERROR;

      stMsg.eType                             := E_MessageType.eMessageError;
      stMsg.eDevice                           := e_Device.Device_MainAxis;
      stMsg.eSubdevice                        := e_SubDevice.MainInit;
      stMsg.iErrorNumber                      := GVL_AXIS.Control[nAxisInit].ErrorId;

      stMsg.sText                             := concat('MAIN_AXIS.eInit ERROR at Index: ', TO_STRING(nAxisInit));
      f_MessageSet(stMsg);

    ELSIF (GVL_AXIS.State[nAxisInit].eState = E_AXIS_STATE.AXIS_INIT + E_PROGRESS.PROGRESS_DONE)
    THEN
      eInit                                   := E_PROGRESS.PROGRESS_CHECK;
    END_IF
  //-----------------------------------------------------------------------------
  //-----------------------------------------------------------------------------
  E_PROGRESS.PROGRESS_CHECK:
    IF NOT (nAxisInit > PLC_CONSTANT.MAX_AXIS-1)
    THEN
      nAxisInit                               := nAxisInit + 1;
      eInit                                   := E_PROGRESS.PROGRESS_PREPARE;

    ELSE
      eInit                                   := E_PROGRESS.PROGRESS_OCCUPIED;

      stMsg.eType                             := E_MessageType.eMessageInfo;
      stMsg.eDevice                           := e_Device.Device_MainAxis;
      stMsg.eSubdevice                        := e_SubDevice.MainInit;
      stMsg.iErrorNumber                      := MAX_AXIS;

      stMsg.sText                             := concat('MAIN_AXIS.eInit: ', TO_STRING(E_PROGRESS.PROGRESS_DONE));
      f_MessageSet(stMsg);

      FOR nAxis := 1 TO PLC_CONSTANT.MAX_AXIS
      DO
        GVL_MSG_AXIS.MessageLevelAxisPtp[nAxis]  := GVL_MSG.MessageLevel;
      END_FOR
    END_IF

  E_PROGRESS.PROGRESS_OCCUPIED:
   eInit                                     := E_PROGRESS.PROGRESS_DONE;
END_CASE
//-----------------------------------------------------------------------------------------------------------------
// INIT/
//-----------------------------------------------------------------------------------------------------------------
//-----------------------------------------------------------------------------------------------------------------
//-----------------------------------------------------------------------------------------------------------------
// /cyclic
//-----------------------------------------------------------------------------------------------------------------
IF (eInit <> E_PROGRESS.PROGRESS_ERROR)
THEN
  FOR nAxis := 1 TO PLC_CONSTANT.MAX_AXIS
  DO
      GVL_AXIS.Control[nAxis]();
  END_FOR

  GVL_AXIS.ParameterSelector();
END_IF
//-----------------------------------------------------------------------------------------------------------------
// cyclic/
//-----------------------------------------------------------------------------------------------------------------
//-----------------------------------------------------------------------------------------------------------------
//  /logging
//    - all life is problem solving
//-----------------------------------------------------------------------------------------------------------------
GVL_MSG_AXIS.MotionMessageData.Ctrl           REF= GVL_MSG_AXIS.MotionMessageCtrl;
GVL_MSG_AXIS.MotionMessageData.State          REF= GVL_MSG_AXIS.MotionMessageState;
GVL_MSG_AXIS.MotionMessageData.MessageIndex   REF= GVL_MSG_AXIS.MessageMotionIndex;
GVL_MSG_AXIS.MotionMessageData.ErrorIndex     REF= GVL_MSG_AXIS.MessageMotionError;
GVL_MSG_AXIS.MotionMessageData.DirRoot        :=   ADR(GVL_MSG_AXIS.LOG_DIR);
GVL_MSG_AXIS.MotionMessageData.FileRoot       :=   ADR(GVL_MSG_AXIS.LOG_FILE);
GVL_MSG_AXIS.MotionMessageData.MsgList        :=   ADR(GVL_MSG_AXIS.MotionMessages);
GVL_MSG_AXIS.MotionMessageData.LocalTime      :=   ADR(GVL_MSG_AXIS.dtLocalTime);
GVL_MSG_AXIS.MotionMessageData();               

eMsgState                                     :=   f_GetState   (GVL_MSG_AXIS.MotionMessageState.State);
eMsgProgress                                  :=   f_GetProgress(GVL_MSG_AXIS.MotionMessageState.State);

CASE eMsgState
OF
  E_MESSAGE_STATE.MSG_STATE_NULL:
    CASE eMsgProgress
    OF
      E_PROGRESS.PROGRESS_INVALID,
      E_PROGRESS.PROGRESS_DONE:
        IF (GVL_MSG_AXIS.MessageMotionIndex > GVL_MSG.MAX_MESSAGE/100) OR
           (GVL_MSG_AXIS.MessageMotionError > 0)
        THEN
          GVL_MSG_AXIS.MotionMessageCtrl.Cmd  := E_MESSAGE_CTRL.MSG_CTRL_WRITE;
        ELSE
          tonIdleWriteMotion(IN := TRUE, PT:= tIdleWriteMotion);
          IF (tonIdleWriteMotion.Q)
          THEN
            GVL_MSG_AXIS.MotionMessageCtrl.Cmd:= E_MESSAGE_CTRL.MSG_CTRL_WRITE;
          END_IF
        END_IF
    END_CASE

  E_MESSAGE_STATE.MSG_STATE_WRITE:
    CASE eMsgProgress
    OF
      E_PROGRESS.PROGRESS_ERROR,
      E_PROGRESS.PROGRESS_DONE:
        tonIdleWriteMotion(IN := FALSE, PT:= tIdleWriteMotion);
        GVL_MSG_AXIS.MotionMessageCtrl.Cmd    := E_MESSAGE_CTRL.MSG_CTRL_NULL;
    END_CASE

ELSE
    CASE eMsgProgress
    OF
      E_PROGRESS.PROGRESS_DONE:
        GVL_MSG_AXIS.MotionMessageCtrl.Cmd    := E_MESSAGE_CTRL.MSG_CTRL_NULL;
    END_CASE
END_CASE
//-----------------------------------------------------------------------------------------------------------------
//  logging/
//-----------------------------------------------------------------------------------------------------------------
//-----------------------------------------------------------------------------------------------------------------
//-----------------------------------------------------------------------------------------------------------------
//  /Metrics
//-----------------------------------------------------------------------------------------------------------------
GVL_MSG_AXIS.MetricMessageData.Ctrl           REF= GVL_MSG_AXIS.MetricMessageCtrl;
GVL_MSG_AXIS.MetricMessageData.State          REF= GVL_MSG_AXIS.MetricMessageState;

GVL_MSG_AXIS.MetricMessageData.MessageIndex   REF= GVL_MSG_AXIS.MessageMetricIndex;
GVL_MSG_AXIS.MetricMessageData.ErrorIndex     REF= GVL_MSG_AXIS.MessageMetricError;

GVL_MSG_AXIS.MetricMessageData.DirRoot        :=   ADR(GVL_MSG_AXIS.LOG_DIR);
GVL_MSG_AXIS.MetricMessageData.FileRoot       :=   ADR(GVL_MSG_AXIS.LOG_FILE_METRIC);

GVL_MSG_AXIS.MetricMessageData.MsgList        :=   ADR(GVL_MSG_AXIS.MetricMessages);
GVL_MSG_AXIS.MetricMessageData.LocalTime      :=   ADR(GVL_MSG_AXIS.dtLocalTime);

GVL_MSG_AXIS.MetricMessageData();

eMtrState                                     := f_GetState   (GVL_MSG_AXIS.MetricMessageState.State);
eMtrProgress                                  := f_GetProgress(GVL_MSG_AXIS.MetricMessageState.State);

CASE eMtrState
OF
  E_MESSAGE_STATE.MSG_STATE_NULL:
    CASE eMtrProgress
    OF
      E_PROGRESS.PROGRESS_INVALID:
        IF (GVL_MSG_AXIS.MessageMetricIndex > GVL_MSG.MAX_MESSAGE/100) OR
           (GVL_MSG_AXIS.MessageMetricError > 0)
        THEN
          GVL_MSG_AXIS.MetricMessageCtrl.Cmd  := E_MESSAGE_CTRL.MSG_CTRL_WRITE;
        ELSE
          tonIdleWriteMetric(IN := TRUE, PT:= tIdleWriteMetric);
          IF (tonIdleWriteMetric.Q)
          THEN
            GVL_MSG_AXIS.MetricMessageCtrl.Cmd:= E_MESSAGE_CTRL.MSG_CTRL_WRITE;
          END_IF
        END_IF
    END_CASE

  E_MESSAGE_STATE.MSG_STATE_WRITE:
    CASE eMtrProgress
    OF
      E_PROGRESS.PROGRESS_ERROR,
      E_PROGRESS.PROGRESS_DONE:
        tonIdleWriteMetric(IN := FALSE, PT:= tIdleWriteMetric);
        GVL_MSG_AXIS.MetricMessageCtrl.Cmd    := E_MESSAGE_CTRL.MSG_CTRL_NULL;
    END_CASE
ELSE
    CASE eMtrProgress
    OF
      E_PROGRESS.PROGRESS_DONE:
        GVL_MSG_AXIS.MetricMessageCtrl.Cmd    := E_MESSAGE_CTRL.MSG_CTRL_NULL;
    END_CASE
END_CASE
//-----------------------------------------------------------------------------------------------------------------
//  Metrics/
//-----------------------------------------------------------------------------------------------------------------
//-----------------------------------------------------------------------------------------------------------------

END_PROGRAM

// ---- _types/f_GetProgress.TcPOU
// global function to extract e_progress from combined value
FUNCTION f_GetProgress : uint
VAR_INPUT
  state     : UINT;
END_VAR
VAR
  nP        : uint;
END_VAR


nP := state / E_PROGRESS.PROGRESS_INIT;

f_GetProgress := nP * E_PROGRESS.PROGRESS_INIT;

END_FUNCTION

// ---- NCI/NCI.TcPOU
PROGRAM NCI
VAR
  eInit                     : E_PROGRESS;

  nChn,
  nChnInit,
  nAxis,
  nAxisInit                 : UINT;

  stMsg                     : ST_Message;
END_VAR

//-----------------------------------------------------------------------------------------------------------------
// check if compiler define is present [PLC_STATE_DRIVE/CompilerDefines/Manual: NCI]
// see PLC_CONSTANT for conditional pragma
//-----------------------------------------------------------------------------------------------------------------
IF NOT PLC_CONSTANT.NCI_ACTIVE THEN eInit   := E_PROGRESS.PROGRESS_NOT_EXIST; RETURN; END_IF
//-----------------------------------------------------------------------------------------------------------------
//-----------------------------------------------------------------------------------------------------------------
// check for MAIN.eInit
//-----------------------------------------------------------------------------------------------------------------
IF NOT (MAIN_AXIS.eInit = E_PROGRESS.PROGRESS_DONE) THEN eInit   := E_PROGRESS.PROGRESS_INVALID; RETURN; END_IF
//-----------------------------------------------------------------------------------------------------------------
//-----------------------------------------------------------------------------------------------------------------
// /assign dataflow
//-----------------------------------------------------------------------------------------------------------------
FOR nChn := 1 TO MAX_NCI_CH
DO
  // NCI axis configuration --> NC AxisId used
  GVL_NCI.NciCtrl[nChn].ItfChannel.CfgAxes          := ADR(GVL_NCI.AxisConfig[nChn]);

  // R Parameter properties
  GVL_NCI.NciCtrl[nChn].ItfChannel.R_ParameterRead  := ADR(GVL_NCI.R_ParameterRead[nChn]);
  GVL_NCI.NciCtrl[nChn].ItfChannel.R_ParameterWrite := ADR(GVL_NCI.R_ParameterWrite[nChn]);

  // ProgName for channel
  GVL_NCI.NciCtrl[nChn].ItfChannel.Prog             := GVL_NCI.ChannelCtrl[nChn].sProgramName;

  // check REAL value to avoid exception
  IF NOT IsFinite(F_Real(GVL_NCI.ChannelCtrl[nChn].rOverride))
  THEN
    GVL_NCI.NciCtrl[nChn].ItfChannel.Override       := 0.0;
  ELSE
    GVL_NCI.NciCtrl[nChn].ItfChannel.Override       := GVL_NCI.ChannelCtrl[nChn].rOverride;
  END_IF

  // command and state structure assignement
  GVL_NCI.NciCtrl[nChn].ChnCtrl                     := ADR(GVL_NCI.ChannelCtrl[nChn]);
  GVL_NCI.NciCtrl[nChn].ChnState                    := ADR(GVL_NCI.ChannelState[nChn]);
END_FOR
//-----------------------------------------------------------------------------------------------------------------
// assign dataflow/
//-----------------------------------------------------------------------------------------------------------------
//-----------------------------------------------------------------------------------------------------------------
// /INIT
//-----------------------------------------------------------------------------------------------------------------
CASE eInit
OF
  E_PROGRESS.PROGRESS_INVALID:
    FOR nChn := 1 TO MAX_NCI_CH
    DO
      GVL_MSG_AXIS.MessageLevelNciChn[nChn]         := E_MessageType.eMessageVerbose;//GVL_MSG.MessageLevel;
    END_FOR
    nChnInit                                        := 1;
    eInit                                           := E_PROGRESS.PROGRESS_INIT;
  //-----------------------------------------------------------------------------
  //-----------------------------------------------------------------------------
  E_PROGRESS.PROGRESS_INIT:
    stMsg.eType                                     := E_MessageType.eMessageInfo;
    stMsg.eDevice                                   := e_Device.Device_Nci;
    stMsg.eSubdevice                                := e_SubDevice.MainInit;
    stMsg.iErrorNumber                              := MAX_AXIS;
    stMsg.sText                                     := concat('NCI.eInit: ', TO_STRING(eInit));
    f_MessageSet(stMsg);                          

    eInit                                           := E_PROGRESS.PROGRESS_BUSY;
  //-----------------------------------------------------------------------------
  //-----------------------------------------------------------------------------
  E_PROGRESS.PROGRESS_BUSY:
    eInit                                           := E_PROGRESS.PROGRESS_PREPARE;
  //-----------------------------------------------------------------------------
  //-----------------------------------------------------------------------------
  E_PROGRESS.PROGRESS_PREPARE:
    stMsg.eType                                     := E_MessageType.eMessageVerbose;
    stMsg.eDevice                                   := e_Device.Device_Nci;
    stMsg.eSubdevice                                := e_SubDevice.NciStartUp;
    stMsg.iErrorNumber                              := nChnInit;
    stMsg.sText                                     := concat('nChnInit: ', TO_STRING(nChnInit));

    IF (GVL_MSG_AXIS.MessageLevelNciChn[nChnInit] = E_MessageType.eMessageVerbose)
    THEN
      f_MessageSet(stMsg);
    END_IF

    GVL_NCI.ChannelCtrl[nChnInit].eCmd              := E_NCI_CTRL.NULL;
    eInit                                           := E_PROGRESS.PROGRESS_STARTUP;
  //-----------------------------------------------------------------------------
  //-----------------------------------------------------------------------------
  E_PROGRESS.PROGRESS_STARTUP:
    GVL_NCI.ChannelCtrl[nChnInit].eCmd              := E_NCI_CTRL.INIT;

    IF (GVL_NCI.ChannelState[nChnInit].eState = E_NCI_STATE.INIT + E_PROGRESS.PROGRESS_ERROR)
    THEN
      eInit                                         := E_PROGRESS.PROGRESS_ERROR;

      stMsg.eType                                   := E_MessageType.eMessageError;
      stMsg.eDevice                                 := e_Device.Device_Nci;
      stMsg.eSubdevice                              := e_SubDevice.NciStartUp;
      stMsg.iErrorNumber                            := nChnInit;
      stMsg.sText                                   := concat('NCI.eInit ERROR at Index: ', TO_STRING(nChnInit));
      f_MessageSet(stMsg);

    ELSIF (GVL_NCI.ChannelState[nChnInit].eState = E_NCI_STATE.INIT + E_PROGRESS.PROGRESS_DONE)
    THEN
      eInit                                         := E_PROGRESS.PROGRESS_CHECK;
    END_IF
  //-----------------------------------------------------------------------------
  //-----------------------------------------------------------------------------
  E_PROGRESS.PROGRESS_CHECK:
    IF (nChnInit > PLC_CONSTANT.MAX_NCI_CH-1)
    THEN
      eInit                                         := E_PROGRESS.PROGRESS_DONE;

      stMsg.eType                                   := E_MessageType.eMessageInfo;
      stMsg.eDevice                                 := e_Device.Device_Nci;
      stMsg.eSubdevice                              := e_SubDevice.NciStartUp;
      stMsg.iErrorNumber                            := MAX_NCI_CH;
      stMsg.sText                                   := concat('NCI.eInit: ', TO_STRING(eInit));
      f_MessageSet(stMsg);

      FOR nChn := 1 TO MAX_NCI_CH
      DO
        GVL_MSG_AXIS.MessageLevelNciChn[nChn]       := GVL_MSG_AXIS.MessageLevel;
      END_FOR

    ELSE
      nChnInit                                      := nChnInit + 1;
      eInit                                         := E_PROGRESS.PROGRESS_PREPARE;
    END_IF
END_CASE
//-----------------------------------------------------------------------------------------------------------------
// INIT/
//-----------------------------------------------------------------------------------------------------------------
//-----------------------------------------------------------------------------------------------------------------
//-----------------------------------------------------------------------------------------------------------------
// /CYCLE
//-----------------------------------------------------------------------------------------------------------------
FOR nChn := 1 TO MAX_NCI_CH
DO
  // call nci channel controller
  GVL_NCI.NciCtrl[nChn].Cycle();

  GVL_NCI.ProgramNameActive[nChn]                   := GVL_NCI.NciCtrl[nChn].ItfChannel.GetLoadedProg();
  GVL_NCI.ChannelState[nChn].sProgramNameActive     := GVL_NCI.ProgramNameActive[nChn];
  GVL_NCI.NciCtrl[nChn].M_FunctionScope             := ADR(GVL_NCI.M_FunctionCyclic[nChn]);
END_FOR
//-----------------------------------------------------------------------------------------------------------------
// CYCLE/
//-----------------------------------------------------------------------------------------------------------------
//-----------------------------------------------------------------------------------------------------------------

END_PROGRAM

// ---- FLYING_SAW/FLYING_SAW.TcPOU
PROGRAM FLYING_SAW
VAR
  eInit             : E_PROGRESS;

  nAxisInit,
  nAxis             : UINT;

  stMsg             : ST_Message;
END_VAR

//-----------------------------------------------------------------------------------------------------------------
// check if compiler define is present [PLC_MOTION/CompilerDefines/Manual: SAW]
// see PLC_CONSTANT for conditional pragma
//-----------------------------------------------------------------------------------------------------------------
IF NOT PLC_CONSTANT.FLY_SAW_ACTIVE THEN eInit := E_PROGRESS.PROGRESS_NOT_EXIST; RETURN; END_IF
//-----------------------------------------------------------------------------------------------------------------
//-----------------------------------------------------------------------------------------------------------------
// check for MAIN.eInit
//-----------------------------------------------------------------------------------------------------------------
IF NOT (MAIN_AXIS.eInit = E_PROGRESS.PROGRESS_DONE) THEN eInit   := E_PROGRESS.PROGRESS_INVALID; RETURN; END_IF
//-----------------------------------------------------------------------------------------------------------------
//-----------------------------------------------------------------------------------------------------------------
// /assign dataflow
//-----------------------------------------------------------------------------------------------------------------
FOR nAxis := 1 TO PLC_CONSTANT.MAX_AXIS
DO
  GVL_FLYING_SAW.Control[nAxis].AxisIndex     := nAxis;
  GVL_FLYING_SAW.Control[nAxis].AxisModulo    := GVL_FLYING_SAW.Data[nAxis].rModulo;
  GVL_FLYING_SAW.Control[nAxis].MessageLevel  := GVL_MSG_AXIS.MessageLevelAxisFly[nAxis];
  GVL_FLYING_SAW.Control[nAxis].ItfMcAxes     := GVL_AXIS.ItfMcAxis;

  GVL_FLYING_SAW.Control[nAxis].AxisCtrl      := ADR(GVL_FLYING_SAW.Ctrl);
  GVL_FLYING_SAW.Control[nAxis].AxisState     := ADR(GVL_FLYING_SAW.State);
  GVL_FLYING_SAW.Control[nAxis].GearData      := ADR(GVL_FLYING_SAW.Data);
  GVL_FLYING_SAW.Control[nAxis].Options       := ADR(GVL_FLYING_SAW.Options);
  GVL_FLYING_SAW.Control[nAxis].MoveData      := ADR(GVL_AXIS.Data);
 END_FOR
//-----------------------------------------------------------------------------------------------------------------
// assign dataflow/
//-----------------------------------------------------------------------------------------------------------------
//-----------------------------------------------------------------------------------------------------------------
// /INIT
//-----------------------------------------------------------------------------------------------------------------
CASE eInit
OF
  E_PROGRESS.PROGRESS_INVALID:
    nAxisInit                                 := 1;
    eInit                                     := E_PROGRESS.PROGRESS_INIT;

    FOR nAxis := 1 TO PLC_CONSTANT.MAX_AXIS
    DO
      GVL_MSG_AXIS.MessageLevelAxisFly[nAxis] := GVL_MSG_AXIS.MessageLevel;
    END_FOR
  //-----------------------------------------------------------------------------
  //-----------------------------------------------------------------------------
  E_PROGRESS.PROGRESS_INIT:
    stMsg.eType                               := E_MessageType.eMessageInfo;
    stMsg.eDevice                             := e_Device.Device_FlyingSaw;
    stMsg.eSubdevice                          := e_SubDevice.FlyingSawStartUp;
    stMsg.iErrorNumber                        := MAX_AXIS;
    stMsg.sText                               := concat('FLYING_SAW.eInit: ', TO_STRING(eInit));
    f_MessageSet(stMsg);

    eInit                                     := E_PROGRESS.PROGRESS_BUSY;
  //-----------------------------------------------------------------------------
  //-----------------------------------------------------------------------------
  E_PROGRESS.PROGRESS_BUSY:
    eInit                                     := E_PROGRESS.PROGRESS_PREPARE;
  //-----------------------------------------------------------------------------
  //-----------------------------------------------------------------------------
  E_PROGRESS.PROGRESS_PREPARE:
    stMsg.eType                               := E_MessageType.eMessageVerbose;
    stMsg.eDevice                             := e_Device.Device_FlyingSaw;
    stMsg.eSubdevice                          := e_SubDevice.FlyingSawStartUp;
    stMsg.iErrorNumber                        := nAxisInit;
    stMsg.sText                               := concat('AxisInit: ', TO_STRING(nAxisInit));

    IF (GVL_MSG_AXIS.MessageLevelAxisFly[nAxisInit] = E_MessageType.eMessageVerbose)
    THEN
      f_MessageSet(stMsg);
    END_IF

    GVL_FLYING_SAW.Ctrl[nAxisInit].eCmd       := E_AXIS_CTRL.AXIS_NULL;
    eInit                                     := E_PROGRESS.PROGRESS_STARTUP;
  //-----------------------------------------------------------------------------
  //-----------------------------------------------------------------------------
  E_PROGRESS.PROGRESS_STARTUP:
    GVL_FLYING_SAW.Ctrl[nAxisInit].eCmd       := E_AXIS_CTRL.AXIS_INIT;

    IF (GVL_FLYING_SAW.State[nAxisInit].eState = E_AXIS_STATE.AXIS_INIT + E_PROGRESS.PROGRESS_ERROR)
    THEN
      eInit                                   := E_PROGRESS.PROGRESS_ERROR;

    ELSIF (GVL_FLYING_SAW.State[nAxisInit].eState = E_AXIS_STATE.AXIS_INIT + E_PROGRESS.PROGRESS_DONE)
    THEN
      eInit                                   := E_PROGRESS.PROGRESS_CHECK;
    END_IF
  //-----------------------------------------------------------------------------
  //-----------------------------------------------------------------------------
  E_PROGRESS.PROGRESS_CHECK:
    IF (nAxisInit > PLC_CONSTANT.MAX_AXIS-1)
    THEN
      eInit                                   := E_PROGRESS.PROGRESS_DONE;

      stMsg.eType                             := E_MessageType.eMessageInfo;
      stMsg.eDevice                           := e_Device.Device_FlyingSaw;
      stMsg.eSubdevice                        := e_SubDevice.FlyingSawStartUp;
      stMsg.iErrorNumber                      := MAX_AXIS;

      stMsg.sText                             := concat('FLYING_SAW.eInit: ', TO_STRING(eInit));
      f_MessageSet(stMsg);
    ELSE
      nAxisInit                               := nAxisInit + 1;
      eInit                                   := E_PROGRESS.PROGRESS_PREPARE;
    END_IF
END_CASE
//-----------------------------------------------------------------------------------------------------------------
// INIT
//-----------------------------------------------------------------------------------------------------------------
//-----------------------------------------------------------------------------------------------------------------
// /cyclic
//-----------------------------------------------------------------------------------------------------------------
IF (eInit <> E_PROGRESS.PROGRESS_ERROR)
THEN
  FOR nAxis := 1 TO PLC_CONSTANT.MAX_AXIS
  DO
      GVL_FLYING_SAW.Control[nAxis].Cycle();
  END_FOR
END_IF
//-----------------------------------------------------------------------------------------------------------------
// cyclic/
//-----------------------------------------------------------------------------------------------------------------

END_PROGRAM

// ---- NC_PTP/class/FB_McAxisBase.TcPOU
FUNCTION_BLOCK ABSTRACT FB_McAxisBase  IMPLEMENTS I_McAxis
VAR
  _AxisRef                      : REFERENCE TO Tc2_MC2.AXIS_REF;
  _pCalibrationCam              : POINTER TO BOOL;

  _nErrorId                     : UDINT; // datafield for MC error

  _MessageLevel                 : E_MessageType;

  // MC_Power inputs for feed fwd, feed bwd, override
  _bEnablePositive              : BOOL  := TRUE;
  _bEnableNegative              : BOOL  := TRUE;
  _rAxisOverride                : LREAL := 100.0;

  _rValueParameterRead          : LREAL;
  _fbReadParameter              : Tc2_MC2.MC_ReadParameter;
  _fbWriteParameter             : Tc2_MC2.MC_WriteParameter;
  _fbWriteParameterPersist      : Tc2_MC2.MC_WriteParameterPersistent;

  // last target position datafield
  _rLastTargetPosition          : LREAL;

  // name and encoder type are read by ADSREAD instance from NC
  _sAxisName                    : STRING(30) := 'NO NAME'; // AxisName is limited to 30 chars, IdxGrp := 4000 + _AxisRef.NcToPlc.AxisId, IdxOffs := 16#02
  _sEncoderType                 : STRING(30) := 'NO TYPE';
  _nEncoderType                 : UDINT;
  _eEncoderType                 : E_AxisEncoderType;

  // Motion Control FB Instances
  _fbPower                      : Tc2_MC2.MC_Power;
  _fbReset                      : Tc2_MC2.MC_Reset;
  _fbHalt                       : Tc2_MC2.MC_Halt;
  _fbStop                       : Tc2_MC2.MC_Stop;
  _fbHome                       : Tc2_MC2.MC_Home;
  _fbJog                        : Tc2_MC2.MC_Jog;
  _fbMoveToPosition             : Tc2_MC2.MC_MoveAbsolute;
  _fbMoveVelo                   : Tc2_MC2.MC_MoveVelocity;

  // used for buffered moves
  _fbMoveVelocity               : ARRAY[1..2]   OF  Tc2_MC2.MC_MoveVelocity;
  _fbMoveAbsolute               : ARRAY[1..2]   OF  Tc2_MC2.MC_MoveAbsolute;

  // ADS read instance for reading startup information from NC
  _fbADSRead                     : ADSREAD;

  // startup states for getting ADS information from NC
  _nStartUpErrorState,
  _nStartUp                     : DINT := 0;

  _bStartUpError,
  _bStartUp                     : BOOL;

  _rCycleTime                   : LREAL;
  _fbGetCurTaskIndex            : Tc2_System.GETCURTASKINDEX;
END_VAR

PROPERTY AxisEnableNegative : BOOL
GET
AxisEnableNegative := _bEnableNegative;
END_GET
SET
_bEnableNegative := AxisEnableNegative;
END_SET
END_PROPERTY

PROPERTY AxisEnablePositive : BOOL
GET
AxisEnablePositive  := _bEnablePositive;
END_GET
SET
_bEnablePositive := AxisEnablePositive;
END_SET
END_PROPERTY

PROPERTY AxisName : string(30)
GET
AxisName := _sAxisName;
END_GET
END_PROPERTY

PROPERTY AxisRef : reference to AXIS_REF
GET
AxisRef REF= _AxisRef;
END_GET
END_PROPERTY

PROPERTY CalibrationCam : pointer to bool
GET
CalibrationCam  := _pCalibrationCam;
END_GET
SET
_pCalibrationCam := CalibrationCam;
END_SET
END_PROPERTY

METHOD Cycle : E_PROGRESS
VAR_INST
  _eState           : E_PROGRESS;
  _rValue           : LREAL;
  _stMsg            : ST_Message;
END_VAR
IF NOT (__ISVALIDREF(_AxisRef))
THEN
  Cycle                           := E_PROGRESS.PROGRESS_ERROR;
  RETURN;
END_IF

// call cyclic NC interface
_AxisRef();

_fbPower(
        Axis                      := _AxisRef, 
        Enable_Positive           := _bEnablePositive, 
        Enable_Negative           := _bEnableNegative, 
        Override                  := _rAxisOverride);

CASE _eState
OF
  E_PROGRESS.PROGRESS_INVALID:
    _fbGetCurTaskIndex();
    _rCycleTime                   := UDINT_TO_LREAL(_TaskInfo[_fbGetCurTaskIndex.index].CycleTime)/10000.0;

    _eState                       := E_PROGRESS.PROGRESS_BUSY;
END_CASE
CASE _eState
OF
  E_PROGRESS.PROGRESS_BUSY:
    IF (_fbPower.Error) OR
       (_AxisRef.Status.Error)
    THEN
      _eState                     := E_PROGRESS.PROGRESS_ERROR;

      _nErrorId                   := SEL((_fbPower.ErrorID > 0), _AxisRef.NcToPlc.ErrorCode, _fbPower.ErrorID);

      IF (_nErrorId <> _stMsg.iErrorNumber)
      THEN
        _stMsg.eType                := E_MessageType.eMessageError;
        _stMsg.eDevice              := e_Device.Axis + (_AxisRef.NcToPlc.AxisId);;
        _stMsg.eSubdevice           := e_Subdevice.AxisCycle;
        _stMsg.iErrorNumber         := _nErrorId;
  
        _stMsg.sText                := concat(' : ', TO_STRING(_eState));
  
        f_MessageSet(_stMsg);
      END_IF
    ELSE
      _eState                     := E_PROGRESS.PROGRESS_WORKING;
    END_IF
END_CASE
CASE _eState
OF
  E_PROGRESS.PROGRESS_WORKING:
    // rinse, repeat
    _eState                       := E_PROGRESS.PROGRESS_BUSY;
    Cycle                         := E_PROGRESS.PROGRESS_WORKING;
END_CASE
CASE _eState
OF
  E_PROGRESS.PROGRESS_ERROR:
    IF NOT (_fbPower.Error)
    THEN
      _eState                     := E_PROGRESS.PROGRESS_BUSY;
    ELSE
      Cycle                       := E_PROGRESS.PROGRESS_ERROR;
    END_IF
END_CASE
END_METHOD

METHOD Disable : E_PROGRESS
VAR_INPUT
  Execute           : BOOL;
END_VAR
VAR_INST
  _eResult,
  _eState           : E_PROGRESS;
  _rValue           : LREAL;
  _stMsg            : ST_Message;
END_VAR
IF NOT (__ISVALIDREF(_AxisRef)) THEN  Disable  := E_PROGRESS.PROGRESS_ERROR; RETURN; END_IF
IF NOT Execute THEN _eState := E_PROGRESS.PROGRESS_INIT; END_IF

CASE _eState
OF
  E_PROGRESS.PROGRESS_INIT:
    IF Execute 
    THEN
      memset(ADR(_stMsg),0,SIZEOF(_stMsg));
      _nErrorId                     := 0;
      _rValue                       := 0;
      _eState                       := E_PROGRESS.PROGRESS_BUSY;
    END_IF
END_CASE
CASE _eState
OF
  E_PROGRESS.PROGRESS_BUSY:
    _fbPower.Enable                 := FALSE;
    _eResult                        := Reset(FALSE);
    _eState                         := E_PROGRESS.PROGRESS_STARTUP;

  E_PROGRESS.PROGRESS_STARTUP:
    IF _fbPower.Error OR
       _AxisRef.Status.Error
    THEN
      _eState                       := E_PROGRESS.PROGRESS_PREPARE;

      _stMsg.eType                  := E_MessageType.eMessageVerbose;
      _stMsg.eDevice                := E_Device.Axis + (_AxisRef.NcToPlc.AxisId);
      _stMsg.eSubdevice             := e_Subdevice.fbPower;
      _stMsg.iErrorNumber           := 0;

      _stMsg.sText                  := concat('clear error on disable : ', TO_STRING(_eState));

      IF (_MessageLevel = E_MessageType.eMessageVerbose)
      THEN
        f_MessageSet(_stMsg);
      END_IF
    ELSE
      _eState                       := E_PROGRESS.PROGRESS_OCCUPIED;
    END_IF
END_CASE
CASE _eState
OF
  E_PROGRESS.PROGRESS_PREPARE:
    _eResult                        := Reset(TRUE);
    IF (_eResult = E_PROGRESS.PROGRESS_DONE)
    THEN
      _eState                       := E_PROGRESS.PROGRESS_OCCUPIED;

      _stMsg.eType                  := E_MessageType.eMessageVerbose;
      _stMsg.eDevice                := E_Device.Axis + (_AxisRef.NcToPlc.AxisId);
      _stMsg.eSubdevice             := e_Subdevice.fbPower;
      _stMsg.iErrorNumber           := 0;

      _stMsg.sText                  := concat('clear error on disable : ', TO_STRING(_eResult));

      IF (_MessageLevel = E_MessageType.eMessageVerbose)
      THEN
        f_MessageSet(_stMsg);
      END_IF
    END_IF
END_CASE
CASE _eState
OF
  E_PROGRESS.PROGRESS_OCCUPIED:
    IF _AxisRef.Status.Error
    THEN
      _nErrorId                     := _AxisRef.NcToPlc.ErrorCode;
    
      _stMsg.eType                  := E_MessageType.eMessageError;
      _stMsg.eDevice                := e_Device.Axis + (_AxisRef.NcToPlc.AxisId);
      _stMsg.eSubdevice             :=  e_SubDevice.fbPower;
      _stMsg.iErrorNumber           := _nErrorId;

      f_MessageSet(_stMsg);
    
      _eState                       := E_PROGRESS.PROGRESS_ERROR;

    ELSIF NOT _AxisRef.Status.ControlLoopClosed
    THEN
      _eState                       := E_PROGRESS.PROGRESS_WORKING;
    END_IF
END_CASE
CASE _eState
OF
  E_PROGRESS.PROGRESS_WORKING:
    _eResult                        := Reset(FALSE);
    _eState                         := E_PROGRESS.PROGRESS_DONE;

      _stMsg.eType                  := E_MessageType.eMessageVerbose;
      _stMsg.eDevice                := E_Device.Axis + (_AxisRef.NcToPlc.AxisId);
      _stMsg.eSubdevice             := e_Subdevice.fbPower;
      _stMsg.iErrorNumber           := 0;

      _stMsg.sText                  := concat(' : ', TO_STRING(_eState));

      IF (_MessageLevel = E_MessageType.eMessageVerbose)
      THEN
        f_MessageSet(_stMsg);
      END_IF
END_CASE

Disable                             := _eState;
END_METHOD

METHOD Enable : E_PROGRESS
VAR_INPUT
  Execute           : BOOL;
END_VAR
VAR_INST
  _eResult,
  _eState           : E_PROGRESS;
  _rValue           : LREAL;
  _stMsg            : ST_Message;
END_VAR
IF NOT (__ISVALIDREF(_AxisRef)) THEN  Enable  := E_PROGRESS.PROGRESS_ERROR; RETURN; END_IF
IF NOT Execute THEN _eState := E_PROGRESS.PROGRESS_INIT; END_IF

CASE _eState
OF
  E_PROGRESS.PROGRESS_INIT:
    IF Execute 
    THEN
      memset(ADR(_stMsg),0,SIZEOF(_stMsg));
      _nErrorId                     := 0;
      _rValue                       := 0;
      _eState                       := E_PROGRESS.PROGRESS_BUSY;
    END_IF
END_CASE
CASE _eState
OF
  E_PROGRESS.PROGRESS_BUSY:
    _fbPower.Enable                 := TRUE;
    _eResult                        := Reset(FALSE);
    _eState                         := E_PROGRESS.PROGRESS_STARTUP;

  E_PROGRESS.PROGRESS_STARTUP:
    IF _fbPower.Error OR
       _AxisRef.Status.Error
    THEN
      _eState                       := E_PROGRESS.PROGRESS_PREPARE;

      _stMsg.eType                  := E_MessageType.eMessageVerbose;
      _stMsg.eDevice                := E_Device.Axis + (_AxisRef.NcToPlc.AxisId);
      _stMsg.eSubdevice             := e_Subdevice.fbPower;
      _stMsg.iErrorNumber           := 0;

      _stMsg.sText                  := concat('clear error on enable : ', TO_STRING(_eState));

      IF (_MessageLevel = E_MessageType.eMessageVerbose)
      THEN
        f_MessageSet(_stMsg);
      END_IF
    ELSE
      _eState                       := E_PROGRESS.PROGRESS_OCCUPIED;
    END_IF
END_CASE
CASE _eState
OF
  E_PROGRESS.PROGRESS_PREPARE:
    _eResult                        := Reset(TRUE);
    IF (_eResult = E_PROGRESS.PROGRESS_DONE)
    THEN
      _eState                       := E_PROGRESS.PROGRESS_OCCUPIED;
    END_IF
END_CASE
CASE _eState
OF
  E_PROGRESS.PROGRESS_OCCUPIED:
    IF _AxisRef.Status.Error
    THEN
      _nErrorId                     := _AxisRef.NcToPlc.ErrorCode;
    
      _stMsg.eType                  := E_MessageType.eMessageError;
      _stMsg.eDevice                := e_Device.Axis + (_AxisRef.NcToPlc.AxisId);
      _stMsg.eSubdevice             :=  e_SubDevice.fbPower;
      _stMsg.iErrorNumber           := _nErrorId;
    
      f_MessageSet(_stMsg);

      _eState                       := E_PROGRESS.PROGRESS_ERROR;

    ELSIF _AxisRef.Status.ControlLoopClosed
    THEN
      _eState                       := E_PROGRESS.PROGRESS_WORKING;
    END_IF
END_CASE
CASE _eState
OF
  E_PROGRESS.PROGRESS_WORKING:
    _eResult                        := Reset(FALSE);
    _eState                         := E_PROGRESS.PROGRESS_DONE;

      _stMsg.eType                  := E_MessageType.eMessageVerbose;
      _stMsg.eDevice                := E_Device.Axis + (_AxisRef.NcToPlc.AxisId);
      _stMsg.eSubdevice             := e_Subdevice.fbPower;
      _stMsg.iErrorNumber           := 0;

      _stMsg.sText                  := concat(' : ', TO_STRING(_eState));

      IF (_MessageLevel = E_MessageType.eMessageVerbose)
      THEN
        f_MessageSet(_stMsg);
      END_IF
END_CASE

Enable                              := _eState;
END_METHOD

PROPERTY EncoderType : E_AxisEncoderType
GET
EncoderType := _eEncoderType;
END_GET
END_PROPERTY

PROPERTY ErrorId : udint
GET
ErrorId := _nErrorId;
END_GET
END_PROPERTY

METHOD Halt : E_PROGRESS
VAR_INPUT
  Execute           : BOOL;
  Dec               : LREAL;
  Jerk              : LREAL;
END_VAR
VAR_INST
  _eState           : E_PROGRESS;
  _rValue           : LREAL;
  _stMsg            : ST_Message;
END_VAR
IF NOT (__ISVALIDREF(_AxisRef)) THEN  Halt  := E_PROGRESS.PROGRESS_ERROR; RETURN; END_IF
IF NOT Execute THEN _eState := E_PROGRESS.PROGRESS_INIT; END_IF

CASE _eState
OF
  E_PROGRESS.PROGRESS_INIT:
    IF Execute 
    THEN
      memset(ADR(_stMsg),0,SIZEOF(_stMsg));
      _nErrorId                     := 0;
      _rValue                       := 0;
      _eState                       := E_PROGRESS.PROGRESS_BUSY;
    END_IF
END_CASE
CASE _eState
OF
  E_PROGRESS.PROGRESS_BUSY:
    _eState                         := E_PROGRESS.PROGRESS_OCCUPIED;
    _fbHalt(
              Axis                  := _AxisRef, 
              Execute               := FALSE, 
              Deceleration          := Dec, 
              Jerk                  := Jerk, 
              BufferMode            := Tc2_MC2.MC_BufferMode.MC_Aborting);
END_CASE
CASE _eState
OF
  E_PROGRESS.PROGRESS_OCCUPIED:
    _fbHalt(
              Axis                  := _AxisRef, 
              Execute               := TRUE, 
              Deceleration          := Dec, 
              Jerk                  := Jerk, 
              BufferMode            := Tc2_MC2.MC_BufferMode.MC_Aborting);

    IF _fbhalt.Error
    THEN
      _eState                       := E_PROGRESS.PROGRESS_ERROR;
        _nErrorId                   := _fbHalt.ErrorID;

        _stMsg.eType                := E_MessageType.eMessageError;
        _stMsg.eDevice              := e_Device.Axis + (_AxisRef.NcToPlc.AxisId);
        _stMsg.eSubdevice           := e_SubDevice.fbHalt;
        _stMsg.iErrorNumber         := _nErrorId;

        _stMsg.sText                := concat(' : ', TO_STRING(_eState));

        f_MessageSet(_stMsg);

        _fbHalt(
              Axis                  := _AxisRef, 
              Execute               := FALSE);
    ELSE
      IF _fbHalt.Done OR
         _AxisRef.Status.NotMoving
      THEN
        _eState                     := E_PROGRESS.PROGRESS_WORKING;

      ELSIF _fbHalt.CommandAborted
      THEN
        _eState                     := E_PROGRESS.PROGRESS_BUSY;

        _stMsg.eType                := E_MessageType.eMessageWarning;
        _stMsg.eDevice              := E_Device.Axis + (_AxisRef.NcToPlc.AxisId);
        _stMsg.eSubdevice           := e_Subdevice.fbHalt;
        _stMsg.iErrorNumber         := 0;
    
        _stMsg.sText                := concat('command aborted : ', TO_STRING(_eState));

        IF (_MessageLevel > E_MessageType.eMessageError)
        THEN
          f_MessageSet(_stMsg);
        END_IF
      END_IF
    END_IF
END_CASE
CASE _eState
OF
  E_PROGRESS.PROGRESS_WORKING:
    _fbHalt(
              Axis                  := _AxisRef, 
              Execute               := FALSE);

    _eState                         := E_PROGRESS.PROGRESS_DONE;

    _stMsg.eType                    := E_MessageType.eMessageVerbose;
    _stMsg.eDevice                  := E_Device.Axis + (_AxisRef.NcToPlc.AxisId);
    _stMsg.eSubdevice               := e_Subdevice.fbHalt;
    _stMsg.iErrorNumber             := 0;

    _stMsg.sText                    := concat(' : ', TO_STRING(_eState));

    IF (_MessageLevel = E_MessageType.eMessageVerbose)
    THEN
      f_MessageSet(_stMsg);
    END_IF
END_CASE

Halt := _eState;
END_METHOD

METHOD Home : E_PROGRESS
VAR_INPUT
  Execute           : BOOL;
  Position          : LREAL := DEFAULT_HOME_POSITION;
  HomingMode        : Tc2_MC2.MC_HomingMode := MC_DefaultHoming;
  Options           : Tc2_MC2.ST_HomingOptions;
END_VAR
VAR_INST
  _eState           : E_PROGRESS;
  _sValue           : STRING(40);
  _rValue           : LREAL;
  _stMsg            : ST_Message;
END_VAR
IF NOT (__ISVALIDREF(_AxisRef)) THEN  Home  := E_PROGRESS.PROGRESS_ERROR; RETURN; END_IF
IF NOT Execute THEN _eState := E_PROGRESS.PROGRESS_INIT; END_IF

CASE _eState
OF
  E_PROGRESS.PROGRESS_INIT:
    IF Execute 
    THEN
      memset(ADR(_stMsg), 0,SIZEOF(_stMsg));
      memset(ADR(_sValue),0,SIZEOF(_sValue));

      _nErrorId                     := 0;
      _rValue                       := 0;
      _eState                       := E_PROGRESS.PROGRESS_BUSY;

      IF NOT (_pCalibrationCam <> 0) 
      THEN
        _eState                     := E_PROGRESS.PROGRESS_ERROR;
        // prevent page fault
        _sValue                     := 'Pointer to calibration cam not set';

        _nErrorId                   := 666;

        _stMsg.eType                := E_MessageType.eMessageError;
        _stMsg.eDevice              := e_Device.Axis + (_AxisRef.NcToPlc.AxisId);
        _stMsg.eSubdevice           := e_SubDevice.fbHome;
        _stMsg.iErrorNumber         := _nErrorId;
        _stMsg.sText                := _sValue;

        f_MessageSet(_stMsg);
      END_IF
    END_IF
END_CASE
CASE _eState
OF
  E_PROGRESS.PROGRESS_BUSY:
    _eState                         := E_PROGRESS.PROGRESS_OCCUPIED;
    _fbHome(
            Axis                    := _AxisRef, 
            Execute                 := FALSE, 
            Position                := Position, 
            HomingMode              := HomingMode, 
            Options                 := Options, 
            bCalibrationCam         := _pCalibrationCam^);
END_CASE
CASE _eState
OF
  E_PROGRESS.PROGRESS_OCCUPIED:
    _fbHome(
            Execute                 := TRUE, 
            Axis                    := _AxisRef);

    IF _fbHome.Done
    THEN
      _eState                       := E_PROGRESS.PROGRESS_WORKING;
    ELSE
      IF _fbHome.Error
      THEN
        _eState                     := E_PROGRESS.PROGRESS_ERROR;
        _nErrorId                   := _fbHome.ErrorID;

        _stMsg.eType                := E_MessageType.eMessageError;
        _stMsg.eDevice              := e_Device.Axis + (_AxisRef.NcToPlc.AxisId);
        _stMsg.eSubdevice           :=  e_SubDevice.fbHome;
        _stMsg.iErrorNumber         := _nErrorId;

        f_MessageSet(_stMsg);

        _fbHome(
            Execute                 := FALSE, 
            Axis                    := _AxisRef);
      END_IF
    END_IF
END_CASE
CASE _eState
OF
  E_PROGRESS.PROGRESS_WORKING:
    _fbHome(
            Execute                 := FALSE, 
            Axis                    := _AxisRef);

    _eState                         := E_PROGRESS.PROGRESS_DONE;

    _stMsg.eType                    := E_MessageType.eMessageVerbose;
    _stMsg.eDevice                  := E_Device.Axis + (_AxisRef.NcToPlc.AxisId);
    _stMsg.eSubdevice               := e_Subdevice.fbHome;
    _stMsg.iErrorNumber             := 0;

    _stMsg.sText                    := concat(' : ', TO_STRING(_eState));
    IF (_MessageLevel = E_MessageType.eMessageVerbose)
    THEN
      f_MessageSet(_stMsg);
    END_IF
END_CASE

Home                                := _eState;
END_METHOD

PROPERTY LastTargetPosition : LREAL
GET
END_GET
END_PROPERTY

PROPERTY MessageLevel : E_MessageType
SET
_MessageLevel := MessageLevel;
END_SET
END_PROPERTY

METHOD MovePosBuffer : E_PROGRESS
VAR_INPUT
  bEnable          : BOOL;
  Position        : LREAL;
  Vel             : LREAL;
  Acc             : LREAL;
  Dec             : LREAL;
  Jerk            : LREAL;
  BufferMode      : Tc2_MC2.MC_BufferMode;
END_VAR
VAR_INST
  _eState           : E_PROGRESS;
  _rValue           : LREAL;
  _stMsg            : ST_Message;
END_VAR
IF NOT (__ISVALIDREF(_AxisRef)) THEN  MovePosBuffer  := E_PROGRESS.PROGRESS_ERROR; RETURN; END_IF
IF NOT bEnable THEN _eState := E_PROGRESS.PROGRESS_INIT; END_IF

CASE _eState
OF
  E_PROGRESS.PROGRESS_INIT:
    IF bEnable 
    THEN
      memset(ADR(_stMsg),0,SIZEOF(_stMsg));
      _nErrorId                     := 0;
      _rValue                       := Position;

      _eState                       := E_PROGRESS.PROGRESS_BUSY;

      _stMsg.eType                  := E_MessageType.eMessageVerbose;
      _stMsg.eDevice                := e_Device.Axis + (_AxisRef.NcToPlc.AxisId);
      _stMsg.eSubdevice             := e_SubDevice.fbMoveAbsolute1;
      _stMsg.iErrorNumber           := 0;

      _stMsg.sText                  := concat('FB start : ', TO_STRING(_rValue));

      IF (_MessageLevel = E_MessageType.eMessageVerbose)
      THEN
        f_MessageSet(_stMsg);
      END_IF
    END_IF
END_CASE
CASE _eState
OF
  E_PROGRESS.PROGRESS_BUSY:
    _eState                         := E_PROGRESS.PROGRESS_STARTUP;
    _fbMoveAbsolute[1](
                    Axis            := _AxisRef,
                    Execute         := FALSE);

    _fbMoveAbsolute[2](
                    Axis            := _AxisRef,
                    Execute         := FALSE);

END_CASE
CASE _eState
OF
  E_PROGRESS.PROGRESS_STARTUP:
    _fbMoveAbsolute[1](
                    Axis            := _AxisRef, 
                    Execute         := TRUE,
                    Position        := _rValue, 
                    Velocity        := Vel, 
                    Acceleration    := Acc, 
                    Deceleration    := Dec, 
                    Jerk            := Jerk, 
                    BufferMode      := BufferMode);

    _fbMoveAbsolute[2](
                    Axis            := _AxisRef,
                    Execute         := FALSE);

    _rLastTargetPosition            := _fbMoveAbsolute[1].Position;

    IF _fbMoveAbsolute[1].Error
    THEN
      _eState                       := E_PROGRESS.PROGRESS_ERROR;
      _nErrorId                     := _fbMoveAbsolute[1].ErrorID;
    
      _stMsg.eType                  := E_MessageType.eMessageError;
      _stMsg.eDevice                := e_Device.Axis + (_AxisRef.NcToPlc.AxisId);
      _stMsg.eSubdevice             :=  e_SubDevice.fbMoveAbsolute1;
      _stMsg.iErrorNumber           := _nErrorId;
    
      _stMsg.sText                  := concat(' : ', TO_STRING(_eState));
    
      f_MessageSet(_stMsg);

    ELSIF (_fbMoveAbsolute[1].Busy)
    THEN
      _eState                       := E_PROGRESS.PROGRESS_PREPARE;

      _stMsg.eType                  := E_MessageType.eMessageVerbose;
      _stMsg.eDevice                := e_Device.Axis + (_AxisRef.NcToPlc.AxisId);
      _stMsg.eSubdevice             :=  e_SubDevice.fbMoveAbsolute1;
      _stMsg.iErrorNumber           := 0;

      _stMsg.sText                  := concat('FB busy: ', TO_STRING(_eState));

      IF (_MessageLevel = E_MessageType.eMessageVerbose)
      THEN
        f_MessageSet(_stMsg);
      END_IF

    ELSIF (_fbMoveAbsolute[1].CommandAborted)
    THEN
      _eState                       := E_PROGRESS.PROGRESS_PREPARE;

      _stMsg.eType                  := E_MessageType.eMessageVerbose;
      _stMsg.eDevice                := e_Device.Axis + (_AxisRef.NcToPlc.AxisId);
      _stMsg.eSubdevice             :=  e_SubDevice.fbMoveAbsolute1;
      _stMsg.iErrorNumber           := 0;

      _stMsg.sText                  := concat('FB aborted: ', TO_STRING(_eState));

      IF (_MessageLevel = E_MessageType.eMessageVerbose)
      THEN
        f_MessageSet(_stMsg);
      END_IF

    ELSIF (_fbMoveAbsolute[1].Done)
    THEN
      _eState                       := E_PROGRESS.PROGRESS_PREPARE;

      _stMsg.eType                  := E_MessageType.eMessageVerbose;
      _stMsg.eDevice                := e_Device.Axis + (_AxisRef.NcToPlc.AxisId);
      _stMsg.eSubdevice             :=  e_SubDevice.fbMoveAbsolute1;
      _stMsg.iErrorNumber           := 0;

      _stMsg.sText                  := concat('FB done: ', TO_STRING(_eState));

      IF (_MessageLevel = E_MessageType.eMessageVerbose)
      THEN
        f_MessageSet(_stMsg);
      END_IF
    END_IF
END_CASE
CASE _eState
OF
  E_PROGRESS.PROGRESS_PREPARE:
    _fbMoveAbsolute[1](
                    Axis            := _AxisRef);
    _fbMoveAbsolute[2](
                    Axis            := _AxisRef,
                    Execute         := FALSE);

    IF _fbMoveAbsolute[1].Error
    THEN
      _eState                       := E_PROGRESS.PROGRESS_ERROR;
      _nErrorId                     := _fbMoveAbsolute[1].ErrorID;
    
      _stMsg.eType                  := E_MessageType.eMessageError;
      _stMsg.eDevice                := e_Device.Axis + (_AxisRef.NcToPlc.AxisId);
      _stMsg.eSubdevice             :=  e_SubDevice.fbMoveAbsolute1;
      _stMsg.iErrorNumber           := _nErrorId;
    
      _stMsg.sText                  := concat(' : ', TO_STRING(_eState));
    
      f_MessageSet(_stMsg);

    ELSIF (Position <> _rValue)
    THEN
      IF _fbMoveAbsolute[1].Active
      THEN
        _fbMoveAbsolute[1](
                    Axis            := _AxisRef, 
                    Execute         := FALSE);
  
        _eState                       := E_PROGRESS.PROGRESS_CHECK;
  
        _stMsg.eType                  := E_MessageType.eMessageVerbose;
        _stMsg.eDevice                := e_Device.Axis + (_AxisRef.NcToPlc.AxisId);
        _stMsg.eSubdevice             :=  e_SubDevice.fbMoveAbsolute2;
        _stMsg.iErrorNumber           := 0;
  
        _stMsg.sText                  := concat('Position changed: ', TO_STRING(_rValue));
        _stMsg.sText                  := concat(_stMsg.sText        , ' to ');
        _stMsg.sText                  := concat(_stMsg.sText        , TO_STRING(Position));
  
        IF (_MessageLevel = E_MessageType.eMessageVerbose)
        THEN
          f_MessageSet(_stMsg);
        END_IF

        _rValue                       := Position;
      END_IF
    END_IF
END_CASE
CASE _eState
OF
  E_PROGRESS.PROGRESS_CHECK:
    _fbMoveAbsolute[1](
                    Axis            := _AxisRef,
                    Execute         := FALSE);

    _fbMoveAbsolute[2](
                    Axis            := _AxisRef, 
                    Execute         := TRUE,
                    Position        := _rValue, 
                    Velocity        := Vel, 
                    Acceleration    := Acc, 
                    Deceleration    := Dec, 
                    Jerk            := Jerk, 
                    BufferMode      := BufferMode);

    _rLastTargetPosition            := _fbMoveAbsolute[2].Position;

    IF _fbMoveAbsolute[2].Error
    THEN
      _eState                       := E_PROGRESS.PROGRESS_ERROR;
      _nErrorId                     := _fbMoveAbsolute[2].ErrorID;
    
      _stMsg.eType                  := E_MessageType.eMessageError;
      _stMsg.eDevice                := e_Device.Axis + (_AxisRef.NcToPlc.AxisId);
      _stMsg.eSubdevice             :=  e_SubDevice.fbMoveAbsolute2;
      _stMsg.iErrorNumber           := _nErrorId;
    
      _stMsg.sText                  := concat(' : ', TO_STRING(_eState));
    
      f_MessageSet(_stMsg);

    ELSIF (_fbMoveAbsolute[2].Busy)
    THEN
      _eState                       := E_PROGRESS.PROGRESS_OCCUPIED;

      _stMsg.eType                  := E_MessageType.eMessageVerbose;
      _stMsg.eDevice                := e_Device.Axis + (_AxisRef.NcToPlc.AxisId);
      _stMsg.eSubdevice             :=  e_SubDevice.fbMoveAbsolute2;
      _stMsg.iErrorNumber           := 0;

      _stMsg.sText                  := concat('FB busy: ', TO_STRING(_eState));

      IF (_MessageLevel = E_MessageType.eMessageVerbose)
      THEN
        f_MessageSet(_stMsg);
      END_IF

    ELSIF (_fbMoveAbsolute[2].CommandAborted)
    THEN
      _eState                       := E_PROGRESS.PROGRESS_OCCUPIED;

      _stMsg.eType                  := E_MessageType.eMessageVerbose;
      _stMsg.eDevice                := e_Device.Axis + (_AxisRef.NcToPlc.AxisId);
      _stMsg.eSubdevice             :=  e_SubDevice.fbMoveAbsolute2;
      _stMsg.iErrorNumber           := 0;

      _stMsg.sText                  := concat('FB aborted: ', TO_STRING(_eState));

      IF (_MessageLevel = E_MessageType.eMessageVerbose)
      THEN
        f_MessageSet(_stMsg);
      END_IF

    ELSIF (_fbMoveAbsolute[2].Done)
    THEN
      _eState                       := E_PROGRESS.PROGRESS_OCCUPIED;

      _stMsg.eType                  := E_MessageType.eMessageVerbose;
      _stMsg.eDevice                := e_Device.Axis + (_AxisRef.NcToPlc.AxisId);
      _stMsg.eSubdevice             :=  e_SubDevice.fbMoveAbsolute2;
      _stMsg.iErrorNumber           := 0;

      _stMsg.sText                  := concat('FB done: ', TO_STRING(_eState));

      IF (_MessageLevel = E_MessageType.eMessageVerbose)
      THEN
        f_MessageSet(_stMsg);
      END_IF
    END_IF
END_CASE
CASE _eState
OF
  E_PROGRESS.PROGRESS_OCCUPIED:
    _fbMoveAbsolute[1](
                    Axis            := _AxisRef,
                    Execute         := FALSE);

    _fbMoveAbsolute[2](
                    Axis            := _AxisRef);

    IF _fbMoveAbsolute[2].Error
    THEN
      _eState                       := E_PROGRESS.PROGRESS_ERROR;
      _nErrorId                     := _fbMoveAbsolute[2].ErrorID;
    
      _stMsg.eType                  := E_MessageType.eMessageError;
      _stMsg.eDevice                := e_Device.Axis + (_AxisRef.NcToPlc.AxisId);
      _stMsg.eSubdevice             :=  e_SubDevice.fbMoveAbsolute2;
      _stMsg.iErrorNumber           := _nErrorId;
    
      _stMsg.sText                  := concat(' : ', TO_STRING(_eState));
    
      f_MessageSet(_stMsg);

    ELSIF (Position <> _rValue)
    THEN
      IF _fbMoveAbsolute[2].Active
      THEN
        _fbMoveAbsolute[2](Axis       := _AxisRef,
                           Execute    := FALSE);
  
        _eState                       := E_PROGRESS.PROGRESS_STARTUP;
  
        _stMsg.eType                  := E_MessageType.eMessageVerbose;
        _stMsg.eDevice                := e_Device.Axis + (_AxisRef.NcToPlc.AxisId);
        _stMsg.eSubdevice             :=  e_SubDevice.fbMoveAbsolute1;
        _stMsg.iErrorNumber           := 0;
  
        _stMsg.sText                  := concat('Position changed: ', TO_STRING(_rValue));
        _stMsg.sText                  := concat(_stMsg.sText        , ' to ');
        _stMsg.sText                  := concat(_stMsg.sText        , TO_STRING(Position));
  
        IF (_MessageLevel = E_MessageType.eMessageVerbose)
        THEN
          f_MessageSet(_stMsg);
        END_IF
 
        _rValue                       := Position;
      END_IF
    END_IF
END_CASE
CASE _eState
OF
  E_PROGRESS.PROGRESS_INIT,
  E_PROGRESS.PROGRESS_ERROR:
    _fbMoveAbsolute[1](
                    Axis            := _AxisRef,
                    Execute         := FALSE);

    _fbMoveAbsolute[2](
                    Axis            := _AxisRef,
                    Execute         := FALSE);
END_CASE


MovePosBuffer                       := _eState;
END_METHOD

METHOD MoveToPos : E_PROGRESS
VAR_INPUT
  Execute         : BOOL;
  Position        : LREAL;
  Vel             : LREAL;
  Acc             : LREAL;
  Dec             : LREAL;
  Jerk            : LREAL;
  BufferMode      : Tc2_MC2.MC_BufferMode;
END_VAR
VAR_INST
  _eState           : E_PROGRESS;
  _rValue           : LREAL;
  _stMsg            : ST_Message;
END_VAR
IF NOT (__ISVALIDREF(_AxisRef)) THEN  MoveToPos  := E_PROGRESS.PROGRESS_ERROR; RETURN; END_IF
IF NOT Execute THEN _eState := E_PROGRESS.PROGRESS_INIT; END_IF

CASE _eState
OF
  E_PROGRESS.PROGRESS_INIT:
    IF Execute 
    THEN
      memset(ADR(_stMsg),0,SIZEOF(_stMsg));
      _nErrorId                     := 0;
      _rValue                       := 0;
      _eState                       := E_PROGRESS.PROGRESS_BUSY;

      _stMsg.eType                  := E_MessageType.eMessageInfo;
      _stMsg.eDevice                := e_Device.Axis + (_AxisRef.NcToPlc.AxisId);
      _stMsg.eSubdevice             := e_SubDevice.fbMovePtP;
      _stMsg.iErrorNumber           := 0;

      _stMsg.sText                  := concat(' : ', TO_STRING(Position));

      IF (_MessageLevel > E_MessageType.eMessageError)
      THEN
        f_MessageSet(_stMsg);
      END_IF
    END_IF
END_CASE
CASE _eState
OF
  E_PROGRESS.PROGRESS_BUSY:
    _eState                         := E_PROGRESS.PROGRESS_STARTUP;
    _rValue                         := Position;

    _fbMoveToPosition(
                    Axis            := _AxisRef,
                    Execute         := FALSE);
END_CASE
CASE _eState
OF
  E_PROGRESS.PROGRESS_STARTUP:
    _eState                         := E_PROGRESS.PROGRESS_PREPARE;
    _fbMoveToPosition(
                    Axis            := _AxisRef, 
                    Execute         := TRUE,
                    Position        := _rValue, 
                    Velocity        := Vel, 
                    Acceleration    := Acc, 
                    Deceleration    := Dec, 
                    Jerk            := Jerk, 
                    BufferMode      := BufferMode);

    _rLastTargetPosition            := _fbMoveToPosition.Position;
END_CASE
CASE _eState
OF
  E_PROGRESS.PROGRESS_PREPARE:
    _fbMoveToPosition(
                    Axis            := _AxisRef);

    IF (_fbMoveToPosition.Error)
    THEN
      _eState                       := E_PROGRESS.PROGRESS_ERROR;
      _nErrorId                     := _fbMoveToPosition.ErrorID;
    
      _stMsg.eType                  := E_MessageType.eMessageError;
      _stMsg.eDevice                := e_Device.Axis + (_AxisRef.NcToPlc.AxisId);
      _stMsg.eSubdevice             :=  e_SubDevice.fbMovePtP;
      _stMsg.iErrorNumber           := _nErrorId;

      _stMsg.sText                  := concat(' : ', TO_STRING(_eState));
    
      f_MessageSet(_stMsg);

    ELSIF (_fbMoveToPosition.CommandAborted)
    THEN
      _eState                       := E_PROGRESS.PROGRESS_ERROR;
      _nErrorId                     := _fbMoveToPosition.ErrorID;

      _stMsg.eType                  := E_MessageType.eMessageError;
      _stMsg.eDevice                := e_Device.Axis + (_AxisRef.NcToPlc.AxisId);
      _stMsg.eSubdevice             := e_SubDevice.fbMovePtP;
      _stMsg.iErrorNumber           := _nErrorId;

      _stMsg.sText                  := concat('FB aborted: ', TO_STRING(_eState));

      f_MessageSet(_stMsg);

    ELSIF (_fbMoveToPosition.Active)
    THEN
      _eState                       := E_PROGRESS.PROGRESS_OCCUPIED;

      _stMsg.eType                  := E_MessageType.eMessageVerbose;
      _stMsg.eDevice                := e_Device.Axis + (_AxisRef.NcToPlc.AxisId);
      _stMsg.eSubdevice             := e_SubDevice.fbMovePtP;
      _stMsg.iErrorNumber           := 0;

      _stMsg.sText                  := concat('FB active: ', TO_STRING(_eState));

      IF (_MessageLevel = E_MessageType.eMessageVerbose)
      THEN
        f_MessageSet(_stMsg);
      END_IF

    ELSIF (_fbMoveToPosition.Done)
    THEN
      _eState                       := E_PROGRESS.PROGRESS_STILL_WORKING;
    END_IF
END_CASE
CASE _eState
OF
  E_PROGRESS.PROGRESS_OCCUPIED:
    _fbMoveToPosition(
                    Axis            := _AxisRef);

    IF (_fbMoveToPosition.Error)
    THEN
      _eState                       := E_PROGRESS.PROGRESS_ERROR;
      _nErrorId                     := _fbMoveToPosition.ErrorID;
    
      _stMsg.eType                  := E_MessageType.eMessageError;
      _stMsg.eDevice                := e_Device.Axis + (_AxisRef.NcToPlc.AxisId);
      _stMsg.eSubdevice             :=  e_SubDevice.fbMovePtP;
      _stMsg.iErrorNumber           := _nErrorId;

      _stMsg.sText                  := concat(' : ', TO_STRING(_eState));

      f_MessageSet(_stMsg);

    ELSIF (_fbMoveToPosition.CommandAborted)
    THEN
      _eState                       := E_PROGRESS.PROGRESS_ERROR;
      _nErrorId                     := _fbMoveToPosition.ErrorID;
    
      _stMsg.eType                  := E_MessageType.eMessageError;
      _stMsg.eDevice                := e_Device.Axis + (_AxisRef.NcToPlc.AxisId);
      _stMsg.eSubdevice             :=  e_SubDevice.fbMovePtP;
      _stMsg.iErrorNumber           := _nErrorId;

      _stMsg.sText                  := concat('FB aborted : ', TO_STRING(_eState));

      f_MessageSet(_stMsg);

    ELSIF (_fbMoveToPosition.Done)
    THEN
      _eState                       := E_PROGRESS.PROGRESS_STILL_WORKING;
    END_IF
END_CASE
CASE _eState
OF
  E_PROGRESS.PROGRESS_STILL_WORKING:
    _eState                         := E_PROGRESS.PROGRESS_DONE;

    _fbMoveToPosition(
                  Axis              := _AxisRef,
                  Execute           := FALSE);

    _stMsg.eType                    := E_MessageType.eMessageVerbose;
    _stMsg.eDevice                  := e_Device.Axis + (_AxisRef.NcToPlc.AxisId);
    _stMsg.eSubdevice               := e_SubDevice.fbMovePtP;
    _stMsg.iErrorNumber             := 0;

    _stMsg.sText                    := concat(' : ', TO_STRING(_eState));

    IF (_MessageLevel = E_MessageType.eMessageVerbose)
    THEN
      f_MessageSet(_stMsg);
    END_IF
END_CASE

MoveToPos                           := _eState;
END_METHOD

METHOD MoveVelo : E_PROGRESS
VAR_INPUT
  Execute           : BOOL;
  Velocity          : LREAL;
  Acc               : LREAL;
  Dec               : LREAL;
  Jerk              : LREAL;
  Direction         : Tc2_MC2.MC_Direction := MC_Positive_Direction;
  BufferMode        : Tc2_MC2.MC_BufferMode;
END_VAR
VAR_INST
  _eState           : E_PROGRESS;
  _rValue           : LREAL;
  _stMsg            : ST_Message;
END_VAR
IF NOT (__ISVALIDREF(_AxisRef)) THEN  MoveVelo  := E_PROGRESS.PROGRESS_ERROR; RETURN; END_IF
IF NOT Execute THEN _eState := E_PROGRESS.PROGRESS_INIT; END_IF

CASE _eState
OF
  E_PROGRESS.PROGRESS_INIT:
    IF Execute 
    THEN
      memset(ADR(_stMsg),0,SIZEOF(_stMsg));
      _nErrorId                     := 0;
      _rValue                       := Velocity;
      _eState                       := E_PROGRESS.PROGRESS_BUSY;

      _stMsg.eType                  := E_MessageType.eMessageInfo;
      _stMsg.eDevice                := e_Device.Axis + (_AxisRef.NcToPlc.AxisId);
      _stMsg.eSubdevice             := e_SubDevice.fbMoveVelo;
      _stMsg.iErrorNumber           := 0;

      _stMsg.sText                  := concat('FB start : ', TO_STRING(_rValue));

